		// Go back to start
		_inst_intStep := 0;
END_CASE

M_Enable := _bResult;
intEnableStep := _inst_intStep;
END_METHOD

(* This method should explicitly check the enable status of the device.
	Once the enable status is known, this method should return TRUE.
	If this method fails, P_bEnabled should be set to FALSE since the device
	is not absolutely known to still be enabled. *)
METHOD M_GetEnableStatus : BOOL
VAR_OUTPUT
	(* This should return TRUE if the device is explicitly known to be
		enabled, or FALSE otherwise. *)
	bEnabled	: BOOL;
END_VAR
VAR CONSTANT
	_strCOMMAND_NAME : T_MaxString	:= 'GetEnableStatus'; // Name of the API method
	_timeCOMMAND_TIMEOUT : TIME		:= T#5S; // Max time to receive API response
	_strSTART_MSG : T_MaxString		:= 'Getting enable status'; // Prints when method starts
	_strEND_MSG : T_MaxString		:= 'Received enable status'; // Prints when method finishes
	_udintERROR_ID : UDINT			:= E_ApiDeviceError.FailedToGetEnableStatus; // Error ID to set if command fails
	_strERROR_MSG : T_MaxString		:= 'Failed to get enable status!'; // Error message to set if command fails
END_VAR
VAR_INST
	_inst_arrParams: T_ApiParameterList; // Parameters array
	_inst_arrOutputs: T_ApiParameterList; // Outputs array
	_inst_strRet: T_ApiParamValue; // Return string from the router
	_inst_intStep: INT; // Current method step
	_inst_fbParams: FB_ApiParamBuilder; // Parameter builder FB
END_VAR
VAR
	_bComplete: BOOL; // True if the routing finishes
	_intRet: INT; // Return string converted to an integer
	_bResult : BOOL; // Output of the method
	_pArgs: PVOID; // Arguments pointer
END_VAR
_bResult := FALSE;

// Recover from premature stop
bGetEnableStatusBusy := TRUE;
_inst_intStep := intGetEnableStatusStep;

// Steps
CASE _inst_intStep OF
	0: // Wait for no error and router not busy
		IF NOT THIS^.P_bError AND NOT bRouterBusy THEN
			bRouterBusy := TRUE;
			_inst_intStep := _inst_intStep + 10;
		END_IF
		
	10: // Initialize parameters
		THIS^.M_LogMessage(_strSTART_MSG);
		_inst_fbParams.M_ClearParameters();
		_pArgs := _inst_fbParams.M_AddEmptyStruct('args');
		_inst_fbParams.M_OutputToParameterList(_inst_arrParams);
		_inst_intStep := _inst_intStep + 10;
		
	20: // Route the command
		_bComplete := M_RouterHelper(
			_in_strMethodName := _strCOMMAND_NAME, 
			_in_timeTimeout := _timeCOMMAND_TIMEOUT,
			_inout_arrParams := _inst_arrParams,
			_inout_arrOutputs := _inst_arrOutputs,
			_out_strReturnValue=>_inst_strRet);
		
		// If route completed, move to next step
		IF _bComplete THEN
			_inst_intStep := _inst_intStep + 10;
			bRouterBusy := FALSE;
		ELSIF THIS^.P_bError THEN
			_inst_intStep := 0;
			bRouterBusy := FALSE;
		END_IF
		
	30: // Parse results
		_intRet := STRING_TO_INT(_inst_strRet);
		IF _intRet > 0 THEN
			_bResult := TRUE;
			THIS^.M_LogMessage(_strEND_MSG);
			_inst_fbParams.M_LoadFromParameterList(_inst_arrOutputs);
			THIS^.bEnabled := _inst_fbParams.M_ParseBool(
				_inst_fbParams.M_GetParameter('enabled'));
			bEnabled := THIS^.bEnabled;
			
		// Set error if command failed
		ELSE
			THIS^.M_SetError(_udintERROR_ID, _strERROR_MSG);
		END_IF
		
		// Go back to start
		_inst_intStep := 0;
END_CASE

M_GetEnableStatus := _bResult;
intGetEnableStatusStep := _inst_intStep;
END_METHOD

(* This property should be TRUE while any method in this interface is actively
	executing, or FALSE otherwise. *)
PROPERTY P_bEnableBusy : BOOL
GET
P_bEnableBusy := bRouterBusy;
END_GET
END_PROPERTY

(* This should be set to TRUE if M_Enable is successful or M_GetEnableStatus
	determines the device to be enabled, and set to FALSE if M_Disable is
	called at all, M_GetEnableStatus fails, or M_GetEnableStatus determines
	the device to be not enabled. *)
PROPERTY P_bEnabled : BOOL
GET
P_bEnabled := bEnabled;
END_GET
END_PROPERTY

(* This method should explicitly check the power status of the device.
	Once the power status is known, this method should return TRUE.
	If this method fails, P_bPoweredOn should be set to FALSE since the device
	is not absolutely known to still be powered on. *)
METHOD M_GetPowerStatus : BOOL
VAR_OUTPUT
	(* This should return TRUE if the device is explicitly known to be
		powered on, or FALSE otherwise. *)
	bPoweredOn	: BOOL;
END_VAR
VAR CONSTANT
	_strCOMMAND_NAME : T_MaxString	:= 'GetPowerStatus'; // Name of the API method
	_timeCOMMAND_TIMEOUT : TIME		:= T#5S; // Max time to receive API response
	_strSTART_MSG : T_MaxString		:= 'Getting power status'; // Prints when method starts
	_strEND_MSG : T_MaxString		:= 'Received power status'; // Prints when method finishes
	_udintERROR_ID : UDINT			:= E_ApiDeviceError.FailedToGetPowerStatus; // Error ID to set if command fails
	_strERROR_MSG : T_MaxString		:= 'Failed to get power status!'; // Error message to set if command fails
END_VAR
VAR_INST
	_inst_arrParams: T_ApiParameterList; // Parameters array
	_inst_arrOutputs: T_ApiParameterList; // Outputs array
	_inst_strRet: T_ApiParamValue; // Return string from the router
	_inst_intStep: INT; // Current method step
	_inst_fbParams: FB_ApiParamBuilder; // Parameter builder FB
END_VAR
VAR
	_bComplete: BOOL; // True if the routing finishes
	_intRet: INT; // Return string converted to an integer
	_bResult : BOOL; // Output of the method
	_pArgs: PVOID; // Arguments pointer
END_VAR
_bResult := FALSE;

// Recover from premature stop
bGetPowerStatusBusy := TRUE;
_inst_intStep := intGetPowerStatusStep;

// Steps
CASE _inst_intStep OF
	0: // Wait for no error and router not busy
		IF NOT THIS^.P_bError AND NOT bRouterBusy THEN
			bRouterBusy := TRUE;
			_inst_intStep := _inst_intStep + 10;
		END_IF
		
	10: // Initialize parameters
		THIS^.M_LogMessage(_strSTART_MSG);
		_inst_fbParams.M_ClearParameters();
		_pArgs := _inst_fbParams.M_AddEmptyStruct('args');
		_inst_fbParams.M_OutputToParameterList(_inst_arrParams);
		_inst_intStep := _inst_intStep + 10;
		
	20: // Route the command
		_bComplete := M_RouterHelper(
			_in_strMethodName := _strCOMMAND_NAME, 
			_in_timeTimeout := _timeCOMMAND_TIMEOUT,
			_inout_arrParams := _inst_arrParams,
			_inout_arrOutputs := _inst_arrOutputs,
			_out_strReturnValue=>_inst_strRet);
		
		// If route completed, move to next step
		IF _bComplete THEN
			_inst_intStep := _inst_intStep + 10;
			bRouterBusy := FALSE;
		ELSIF THIS^.P_bError THEN
			_inst_intStep := 0;
			bRouterBusy := FALSE;
		END_IF
		
	30: // Parse results
		_intRet := STRING_TO_INT(_inst_strRet);
		IF _intRet > 0 THEN
			_bResult := TRUE;
			THIS^.M_LogMessage(_strEND_MSG);
			_inst_fbParams.M_LoadFromParameterList(_inst_arrOutputs);
			THIS^.bPoweredOn := _inst_fbParams.M_ParseBool(
				_inst_fbParams.M_GetParameter('poweredOn'));
			bPoweredOn := THIS^.bPoweredOn;
			
		// Set error if command failed
		ELSE
			THIS^.M_SetError(_udintERROR_ID, _strERROR_MSG);
		END_IF
		
		// Go back to start
		_inst_intStep := 0;
END_CASE

M_GetPowerStatus := _bResult;
intGetPowerStatusStep := _inst_intStep;
END_METHOD

(* This method should de-energize the device and then return TRUE once
	successful. P_bPoweredOn should be set to FALSE immediately when this is
	called unless the device is explicitly known to still be powered on. *)
METHOD M_PowerOff : BOOL
VAR CONSTANT
	_strCOMMAND_NAME : T_MaxString	:= 'PowerOff'; // Name of the API method
	_timeCOMMAND_TIMEOUT : TIME		:= T#30S; // Max time to receive API response
	_strSTART_MSG : T_MaxString		:= 'Powering off'; // Prints when method starts
	_strEND_MSG : T_MaxString		:= 'Powered off'; // Prints when method finishes
	_udintERROR_ID : UDINT			:= E_ApiDeviceError.FailedToPowerOff; // Error ID to set if command fails
	_strERROR_MSG : T_MaxString		:= 'Failed to power off!'; // Error message to set if command fails
END_VAR
VAR_INST
	_inst_arrParams: T_ApiParameterList; // Parameters array
	_inst_arrOutputs: T_ApiParameterList; // Outputs array
	_inst_strRet: T_ApiParamValue; // Return string from the router
	_inst_intStep: INT; // Current method step
	_inst_fbParams: FB_ApiParamBuilder; // Parameter builder FB
END_VAR
VAR
	_bComplete: BOOL; // True if the routing finishes
	_intRet: INT; // Return string converted to an integer
	_bResult : BOOL; // Output of the method
	_pArgs: PVOID; // Arguments pointer
END_VAR
_bResult := FALSE;

// Recover from premature stop
bPowerOffBusy := TRUE;
_inst_intStep := intPowerOffStep;

// Steps
CASE _inst_intStep OF
	0: // Wait for no error and router not busy
		IF NOT THIS^.P_bError AND NOT bRouterBusy THEN
			bRouterBusy := TRUE;
			_inst_intStep := _inst_intStep + 10;
		END_IF
		
	10: // Initialize parameters
		THIS^.M_LogMessage(_strSTART_MSG);
		_inst_fbParams.M_ClearParameters();
		_pArgs := _inst_fbParams.M_AddEmptyStruct('args');
		_inst_fbParams.M_OutputToParameterList(_inst_arrParams);
		_inst_intStep := _inst_intStep + 10;
		
	20: // Route the command
		_bComplete := M_RouterHelper(
			_in_strMethodName := _strCOMMAND_NAME, 
			_in_timeTimeout := _timeCOMMAND_TIMEOUT,
			_inout_arrParams := _inst_arrParams,
			_inout_arrOutputs := _inst_arrOutputs,
			_out_strReturnValue=>_inst_strRet);
		
		// If route completed, move to next step
		IF _bComplete THEN
			_inst_intStep := _inst_intStep + 10;
			bRouterBusy := FALSE;
		ELSIF THIS^.P_bError THEN
			_inst_intStep := 0;
			bRouterBusy := FALSE;
		END_IF
		
	30: // Parse results
		_intRet := STRING_TO_INT(_inst_strRet);
		IF _intRet > 0 THEN
			_bResult := TRUE;
			THIS^.M_LogMessage(_strEND_MSG);
			_inst_fbParams.M_LoadFromParameterList(_inst_arrOutputs);
			bPoweredOn := FALSE;
			
		// Set error if command failed
		ELSE
			THIS^.M_SetError(_udintERROR_ID, _strERROR_MSG);
		END_IF
		
		// Go back to start
		_inst_intStep := 0;
END_CASE

M_PowerOff := _bResult;
intPowerOffStep := _inst_intStep;
END_METHOD

(* This method should energize the device and then return TRUE and set
	P_bPoweredOn to TRUE once successful. *)
METHOD M_PowerOn : BOOL
VAR CONSTANT
	_strCOMMAND_NAME : T_MaxString	:= 'PowerOn'; // Name of the API method
	_timeCOMMAND_TIMEOUT : TIME		:= T#30S; // Max time to receive API response
	_strSTART_MSG : T_MaxString		:= 'Powering on'; // Prints when method starts
	_strEND_MSG : T_MaxString		:= 'Powered on'; // Prints when method finishes
	_udintERROR_ID : UDINT			:= E_ApiDeviceError.FailedToPowerOn; // Error ID to set if command fails
	_strERROR_MSG : T_MaxString		:= 'Failed to power on!'; // Error message to set if command fails
END_VAR
VAR_INST
	_inst_arrParams: T_ApiParameterList; // Parameters array
	_inst_arrOutputs: T_ApiParameterList; // Outputs array
	_inst_strRet: T_ApiParamValue; // Return string from the router
	_inst_intStep: INT; // Current method step
	_inst_fbParams: FB_ApiParamBuilder; // Parameter builder FB
END_VAR
VAR
	_bComplete: BOOL; // True if the routing finishes
	_intRet: INT; // Return string converted to an integer
	_bResult : BOOL; // Output of the method
	_pArgs: PVOID; // Arguments pointer
END_VAR
_bResult := FALSE;

// Recover from premature stop
bPowerOnBusy := TRUE;
_inst_intStep := intPowerOnStep;

// Steps
CASE _inst_intStep OF
	0: // Wait for no error and router not busy
		IF NOT THIS^.P_bError AND NOT bRouterBusy THEN
			bRouterBusy := TRUE;
			_inst_intStep := _inst_intStep + 10;
		END_IF
		
	10: // Initialize parameters
		THIS^.M_LogMessage(_strSTART_MSG);
		_inst_fbParams.M_ClearParameters();
		_pArgs := _inst_fbParams.M_AddEmptyStruct('args');
		_inst_fbParams.M_AddStructMember(_pArgs, 'scannerName', in_strScannerName);
		_inst_fbParams.M_OutputToParameterList(_inst_arrParams);
		_inst_intStep := _inst_intStep + 10;
		
	20: // Route the command
		_bComplete := M_RouterHelper(
			_in_strMethodName := _strCOMMAND_NAME, 
			_in_timeTimeout := _timeCOMMAND_TIMEOUT,
			_inout_arrParams := _inst_arrParams,
			_inout_arrOutputs := _inst_arrOutputs,
			_out_strReturnValue=>_inst_strRet);
		
		// If route completed, move to next step
		IF _bComplete THEN
			_inst_intStep := _inst_intStep + 10;
			bRouterBusy := FALSE;
		ELSIF THIS^.P_bError THEN
			_inst_intStep := 0;
			bRouterBusy := FALSE;
		END_IF
		
	30: // Parse results
		_intRet := STRING_TO_INT(_inst_strRet);
		IF _intRet > 0 THEN
			_bResult := TRUE;
			THIS^.M_LogMessage(_strEND_MSG);
			_inst_fbParams.M_LoadFromParameterList(_inst_arrOutputs);
			bPoweredOn := TRUE;
			
		// Set error if command failed
		ELSE
			THIS^.M_SetError(_udintERROR_ID, _strERROR_MSG);
		END_IF
		
		// Go back to start
		_inst_intStep := 0;
END_CASE

M_PowerOn := _bResult;
intPowerOnStep := _inst_intStep;
END_METHOD

(* This property should be TRUE while any method in this interface is actively
	executing, or FALSE otherwise. *)
PROPERTY P_bPowerBusy : BOOL
GET
P_bPowerBusy := bRouterBusy;
END_GET
END_PROPERTY

(* This should be set to TRUE if M_PowerOn is successful or if M_GetPowerStatus
	determines that the device is powered on. Otherwise, this should be FALSE. *)
PROPERTY P_bPoweredOn : BOOL
GET
P_bPoweredOn := bPoweredOn;
END_GET
END_PROPERTY

(* This method should explicitly get the current program loaded on the device.
	If the current program is successfully gotten, this method should return
	TRUE and set P_strCurrentProgram and strCurrentProgram to the gotten
	program name. If this method fails, both should be set to empty strings. *)
METHOD M_GetCurrentProgram : BOOL
VAR_OUTPUT
	(* This should be set to the name of the currently loaded program if
		the method was successful, or a blank string otherwise. *)
	strCurrentProgram	: Sensata_Common.T_MaxString;
END_VAR
VAR CONSTANT
	_strCOMMAND_NAME : T_MaxString	:= 'GetCurrentProgram'; // Name of the API method
	_timeCOMMAND_TIMEOUT : TIME		:= T#10S; // Max time to receive API response
	_strSTART_MSG : T_MaxString		:= 'Getting current program'; // Prints when method starts
	_strEND_MSG : T_MaxString		:= 'Received current program'; // Prints when method finishes
	_udintERROR_ID : UDINT			:= E_ApiDeviceError.FailedToGetCurrentProgram; // Error ID to set if command fails
	_strERROR_MSG : T_MaxString		:= 'Failed to get current program!'; // Error message to set if command fails
END_VAR
VAR_INST
	_inst_arrParams: T_ApiParameterList; // Parameters array
	_inst_arrOutputs: T_ApiParameterList; // Outputs array
	_inst_strRet: T_ApiParamValue; // Return string from the router
	_inst_intStep: INT; // Current method step
	_inst_fbParams: FB_ApiParamBuilder; // Parameter builder FB
END_VAR
VAR
	_bComplete: BOOL; // True if the routing finishes
	_intRet: INT; // Return string converted to an integer
	_bResult : BOOL; // Output of the method
	_pArgs: PVOID; // Arguments pointer
END_VAR
_bResult := FALSE;

// Recover from premature stop
bGetCurrentProgramBusy := TRUE;
_inst_intStep := intGetCurrentProgramStep;

// Steps
CASE _inst_intStep OF
	0: // Wait for no error and router not busy
		IF NOT THIS^.P_bError AND NOT bRouterBusy THEN
			bRouterBusy := TRUE;
			_inst_intStep := _inst_intStep + 10;
		END_IF
		
	10: // Initialize parameters
		THIS^.M_LogMessage(_strSTART_MSG);
		_inst_fbParams.M_ClearParameters();
		_pArgs := _inst_fbParams.M_AddEmptyStruct('args');
		_inst_fbParams.M_OutputToParameterList(_inst_arrParams);
		_inst_intStep := _inst_intStep + 10;
		
	20: // Route the command
		_bComplete := M_RouterHelper(
			_in_strMethodName := _strCOMMAND_NAME, 
			_in_timeTimeout := _timeCOMMAND_TIMEOUT,
			_inout_arrParams := _inst_arrParams,
			_inout_arrOutputs := _inst_arrOutputs,
			_out_strReturnValue=>_inst_strRet);
		
		// If route completed, move to next step
		IF _bComplete THEN
			_inst_intStep := _inst_intStep + 10;
			bRouterBusy := FALSE;
		ELSIF THIS^.P_bError THEN
			_inst_intStep := 0;
			bRouterBusy := FALSE;
		END_IF
		
	30: // Parse results
		_intRet := STRING_TO_INT(_inst_strRet);
		IF _intRet > 0 THEN
			_bResult := TRUE;
			THIS^.M_LogMessage(_strEND_MSG);
			_inst_fbParams.M_LoadFromParameterList(_inst_arrOutputs);
			THIS^.strLoadedProgram := _inst_fbParams.M_ParseString(
				_inst_fbParams.M_GetParameter('programName'));
			strCurrentProgram := THIS^.strLoadedProgram;
			
		// Set error if command failed
		ELSE
			THIS^.M_SetError(_udintERROR_ID, _strERROR_MSG);
		END_IF
		
		// Go back to start
		_inst_intStep := 0;
END_CASE

M_GetCurrentProgram := _bResult;
intGetCurrentProgramStep := _inst_intStep;
END_METHOD

(* This method should explicitly check the program state of the device.
	Once the program state is known, this method should return TRUE and set
	P_enumProgramState and enumProgramState to the relevant E_ProgramState
	value, else it should set both to E_ProgramState.Unknown. *)
METHOD M_GetProgramState : BOOL
VAR_OUTPUT
	(* If the program state is successfully gotten, this should be set to
		the relevant E_ProgramState value. If this method fails, this should
		be set to E_ProgramState.Unknown. *)
	enumProgramState	: Sensata_Common.E_ProgramState;
END_VAR
VAR CONSTANT
	_strCOMMAND_NAME : T_MaxString	:= 'GetControlState'; // Name of the API method
	_timeCOMMAND_TIMEOUT : TIME		:= T#10S; // Max time to receive API response
	_strSTART_MSG : T_MaxString		:= 'Getting program state'; // Prints when method starts
	_strEND_MSG : T_MaxString		:= 'Received program state'; // Prints when method finishes
	_udintERROR_ID : UDINT			:= E_ApiDeviceError.FailedToGetProgramState; // Error ID to set if command fails
	_strERROR_MSG : T_MaxString		:= 'Failed to get program state!'; // Error message to set if command fails
END_VAR
VAR_INST
	_inst_arrParams: T_ApiParameterList; // Parameters array
	_inst_arrOutputs: T_ApiParameterList; // Outputs array
	_inst_strRet: T_ApiParamValue; // Return string from the router
	_inst_intStep: INT; // Current method step
	_inst_fbParams: FB_ApiParamBuilder; // Parameter builder FB
END_VAR
VAR
	_bComplete: BOOL; // True if the routing finishes
	_intRet: INT; // Return string converted to an integer
	_bResult : BOOL; // Output of the method
	_pArgs: PVOID; // Arguments pointer
	dintControlState: DINT; // Current program state
END_VAR
_bResult := FALSE;

// Recover from premature stop
bGetProgramStateBusy := TRUE;
_inst_intStep := intGetProgramStateStep;

// Steps
CASE _inst_intStep OF
	0: // Wait for no error and router not busy
		IF NOT THIS^.P_bError AND NOT bRouterBusy THEN
			bRouterBusy := TRUE;
			_inst_intStep := _inst_intStep + 10;
		END_IF
		
	10: // Initialize parameters
		THIS^.M_LogMessage(_strSTART_MSG);
		_inst_fbParams.M_ClearParameters();
		_pArgs := _inst_fbParams.M_AddEmptyStruct('args');
		_inst_fbParams.M_OutputToParameterList(_inst_arrParams);
		_inst_intStep := _inst_intStep + 10;
		
	20: // Route the command
		_bComplete := M_RouterHelper(
			_in_strMethodName := _strCOMMAND_NAME, 
			_in_timeTimeout := _timeCOMMAND_TIMEOUT,
			_inout_arrParams := _inst_arrParams,
			_inout_arrOutputs := _inst_arrOutputs,
			_out_strReturnValue=>_inst_strRet);
		
		// If route completed, move to next step
		IF _bComplete THEN
			_inst_intStep := _inst_intStep + 10;
			bRouterBusy := FALSE;
		ELSIF THIS^.P_bError THEN
			_inst_intStep := 0;
			bRouterBusy := FALSE;
		END_IF
		
	30: // Parse results
		_intRet := STRING_TO_INT(_inst_strRet);
		IF _intRet > 0 THEN
			_bResult := TRUE;
			THIS^.M_LogMessage(_strEND_MSG);
			_inst_fbParams.M_LoadFromParameterList(_inst_arrOutputs);
			dintControlState := _inst_fbParams.M_ParseInt(_inst_fbParams.M_GetParameter('state'));
			CASE dintControlState OF
				0: enumProgramState := E_ProgramState.Unknown;
				1: enumProgramState := E_ProgramState.Stopped;
				2: enumProgramState := E_ProgramState.Running;
				3: enumProgramState := E_ProgramState.Paused;
			ELSE
				enumProgramState := E_ProgramState.Unknown;
			END_CASE
			THIS^.enumProgramState := enumProgramState;
			
		// Set error if command failed
		ELSE
			THIS^.M_SetError(_udintERROR_ID, _strERROR_MSG);
		END_IF
		
		// Go back to start
		_inst_intStep := 0;
END_CASE

M_GetProgramState := _bResult;
intGetProgramStateStep := _inst_intStep;
END_METHOD

(* This method should load a new program onto the device, and then return TRUE
	once program loading is completed. Once this method begins the program loading
	process, P_strCurrentProgram should be cleared unless it is still explicitly
	known to be loaded. *)
METHOD M_LoadProgram : BOOL
VAR_INPUT
END_VAR
VAR CONSTANT
	_strCOMMAND_NAME : T_MaxString	:= 'LoadProgram'; // Name of the API method
	_timeCOMMAND_TIMEOUT : TIME		:= T#30S; // Max time to receive API response
	_strSTART_MSG : T_MaxString		:= 'Loading program'; // Prints when method starts
	_strEND_MSG : T_MaxString		:= 'Loaded program'; // Prints when method finishes
	_udintERROR_ID : UDINT			:= E_ApiDeviceError.FailedToLoadProgram; // Error ID to set if command fails
	_strERROR_MSG : T_MaxString		:= 'Failed to load program!'; // Error message to set if command fails
END_VAR
VAR_INST
	_inst_arrParams: T_ApiParameterList; // Parameters array
	_inst_arrOutputs: T_ApiParameterList; // Outputs array
	_inst_strRet: T_ApiParamValue; // Return string from the router
	_inst_intStep: INT; // Current method step
	_inst_fbParams: FB_ApiParamBuilder; // Parameter builder FB
END_VAR
VAR
	_bComplete: BOOL; // True if the routing finishes
	_intRet: INT; // Return string converted to an integer
	_bResult : BOOL; // Output of the method
	_pArgs: PVOID; // Arguments pointer
END_VAR
_bResult := FALSE;

// Recover from premature stop
bLoadProgramBusy := TRUE;
_inst_intStep := intLoadProgramStep;

// Steps
CASE _inst_intStep OF
	0: // Wait for no error and router not busy
		IF NOT THIS^.P_bError AND NOT bRouterBusy THEN
			bRouterBusy := TRUE;
			_inst_intStep := _inst_intStep + 10;
		END_IF
		
	10: // Initialize parameters
		THIS^.M_LogMessage(_strSTART_MSG);
		_inst_fbParams.M_ClearParameters();
		_pArgs := _inst_fbParams.M_AddEmptyStruct('args');
		_inst_fbParams.M_AddStructMember(_pArgs, 'filename', in_strProgramName);
		_inst_fbParams.M_OutputToParameterList(_inst_arrParams);
		_inst_intStep := _inst_intStep + 10;
		
	20: // Route the command
		_bComplete := M_RouterHelper(
			_in_strMethodName := _strCOMMAND_NAME, 
			_in_timeTimeout := _timeCOMMAND_TIMEOUT,
			_inout_arrParams := _inst_arrParams,
			_inout_arrOutputs := _inst_arrOutputs,
			_out_strReturnValue=>_inst_strRet);
		
		// If route completed, move to next step
		IF _bComplete THEN
			_inst_intStep := _inst_intStep + 10;
			bRouterBusy := FALSE;
		ELSIF THIS^.P_bError THEN
			_inst_intStep := 0;
			bRouterBusy := FALSE;
		END_IF
		
	30: // Parse results
		_intRet := STRING_TO_INT(_inst_strRet);
		IF _intRet > 0 THEN
			_bResult := TRUE;
			THIS^.M_LogMessage(_strEND_MSG);
			_inst_fbParams.M_LoadFromParameterList(_inst_arrOutputs);
			strLoadedProgram := '';
			
		// Set error if command failed
		ELSE
			THIS^.M_SetError(_udintERROR_ID, _strERROR_MSG);
		END_IF
		
		// Go back to start
		_inst_intStep := 0;
END_CASE

M_LoadProgram := _bResult;
intLoadProgramStep := _inst_intStep;
END_METHOD

(* This program should move to the program state from whatever state it was in
	to the Paused state, and then return TRUE once successful. If the program
	state is Stopped, this method should return TRUE but keep the current state
	as Stopped, since Paused at the beginning at the program is equivalent to
	being Stopped. *)
METHOD M_PauseProgram : BOOL
VAR CONSTANT
	_strCOMMAND_NAME : T_MaxString	:= 'PauseProgram'; // Name of the API method
	_timeCOMMAND_TIMEOUT : TIME		:= T#30S; // Max time to receive API response
	_strSTART_MSG : T_MaxString		:= 'Pausing program'; // Prints when method starts
	_strEND_MSG : T_MaxString		:= 'Paused program'; // Prints when method finishes
	_udintERROR_ID : UDINT			:= E_ApiDeviceError.FailedToPauseProgram; // Error ID to set if command fails
	_strERROR_MSG : T_MaxString		:= 'Failed to pause program!'; // Error message to set if command fails
END_VAR
VAR_INST
	_inst_arrParams: T_ApiParameterList; // Parameters array
	_inst_arrOutputs: T_ApiParameterList; // Outputs array
	_inst_strRet: T_ApiParamValue; // Return string from the router
	_inst_intStep: INT; // Current method step
	_inst_fbParams: FB_ApiParamBuilder; // Parameter builder FB
END_VAR
VAR
	_bComplete: BOOL; // True if the routing finishes
	_intRet: INT; // Return string converted to an integer
	_bResult : BOOL; // Output of the method
	_pArgs: PVOID; // Arguments pointer
END_VAR
_bResult := FALSE;

// Recover from premature stop
bPauseProgramBusy := TRUE;
_inst_intStep := intPauseProgramStep;

// Steps
CASE _inst_intStep OF
	0: // Wait for no error and router not busy
		IF NOT THIS^.P_bError AND NOT bRouterBusy THEN
			bRouterBusy := TRUE;
			_inst_intStep := _inst_intStep + 10;
		END_IF
		
	10: // Initialize parameters
		THIS^.M_LogMessage(_strSTART_MSG);
		_inst_fbParams.M_ClearParameters();
		_pArgs := _inst_fbParams.M_AddEmptyStruct('args');
		_inst_fbParams.M_OutputToParameterList(_inst_arrParams);
		_inst_intStep := _inst_intStep + 10;
		
	20: // Route the command
		_bComplete := M_RouterHelper(
			_in_strMethodName := _strCOMMAND_NAME, 
			_in_timeTimeout := _timeCOMMAND_TIMEOUT,
			_inout_arrParams := _inst_arrParams,
			_inout_arrOutputs := _inst_arrOutputs,
			_out_strReturnValue=>_inst_strRet);
		
		// If route completed, move to next step
		IF _bComplete THEN
			_inst_intStep := _inst_intStep + 10;
			bRouterBusy := FALSE;
		ELSIF THIS^.P_bError THEN
			_inst_intStep := 0;
			bRouterBusy := FALSE;
		END_IF
		
	30: // Parse results
		_intRet := STRING_TO_INT(_inst_strRet);
		IF _intRet > 0 THEN
			_bResult := TRUE;
			THIS^.M_LogMessage(_strEND_MSG);
			_inst_fbParams.M_LoadFromParameterList(_inst_arrOutputs);
			enumProgramState := E_ProgramState.Paused;
			
		// Set error if command failed
		ELSE
			THIS^.M_SetError(_udintERROR_ID, _strERROR_MSG);
		END_IF
		
		// Go back to start
		_inst_intStep := 0;
END_CASE

M_PauseProgram := _bResult;
intPauseProgramStep := _inst_intStep;
END_METHOD

(* This should move the program state from whatever state it is in to the
	Running state, and then return TRUE once successful. Starting from the
	Paused state should always continue execution from whatever point the
	program was at when the program was initially paused. *)
METHOD M_StartProgram : BOOL
VAR CONSTANT
	_strCOMMAND_NAME : T_MaxString	:= 'StartProgram'; // Name of the API method
	_timeCOMMAND_TIMEOUT : TIME		:= T#30S; // Max time to receive API response
	_strSTART_MSG : T_MaxString		:= 'Starting program'; // Prints when method starts
	_strEND_MSG : T_MaxString		:= 'Started program'; // Prints when method finishes
	_udintERROR_ID : UDINT			:= E_ApiDeviceError.FailedToStartProgram; // Error ID to set if command fails
	_strERROR_MSG : T_MaxString		:= 'Failed to start program!'; // Error message to set if command fails
END_VAR
VAR_INST
	_inst_arrParams: T_ApiParameterList; // Parameters array
	_inst_arrOutputs: T_ApiParameterList; // Outputs array
	_inst_strRet: T_ApiParamValue; // Return string from the router
	_inst_intStep: INT; // Current method step
	_inst_fbParams: FB_ApiParamBuilder; // Parameter builder FB
END_VAR
VAR
	_bComplete: BOOL; // True if the routing finishes
	_intRet: INT; // Return string converted to an integer
	_bResult : BOOL; // Output of the method
	_pArgs: PVOID; // Arguments pointer
END_VAR
_bResult := FALSE;

// Recover from premature stop
bStartProgramBusy := TRUE;
_inst_intStep := intStartProgramStep;

// Steps
CASE _inst_intStep OF
	0: // Wait for no error and router not busy
		IF NOT THIS^.P_bError AND NOT bRouterBusy THEN
			bRouterBusy := TRUE;
			_inst_intStep := _inst_intStep + 10;
		END_IF
		
	10: // Initialize parameters
		THIS^.M_LogMessage(_strSTART_MSG);
		_inst_fbParams.M_ClearParameters();
		_pArgs := _inst_fbParams.M_AddEmptyStruct('args');
		_inst_fbParams.M_OutputToParameterList(_inst_arrParams);
		_inst_intStep := _inst_intStep + 10;
		
	20: // Route the command
		_bComplete := M_RouterHelper(
			_in_strMethodName := _strCOMMAND_NAME, 
			_in_timeTimeout := _timeCOMMAND_TIMEOUT,
			_inout_arrParams := _inst_arrParams,
			_inout_arrOutputs := _inst_arrOutputs,
			_out_strReturnValue=>_inst_strRet);
		
		// If route completed, move to next step
		IF _bComplete THEN
			_inst_intStep := _inst_intStep + 10;
			bRouterBusy := FALSE;
		ELSIF THIS^.P_bError THEN
			_inst_intStep := 0;
			bRouterBusy := FALSE;
		END_IF
		
	30: // Parse results
		_intRet := STRING_TO_INT(_inst_strRet);
		IF _intRet > 0 THEN
			_bResult := TRUE;
			THIS^.M_LogMessage(_strEND_MSG);
			_inst_fbParams.M_LoadFromParameterList(_inst_arrOutputs);
			enumProgramState := E_ProgramState.Running;
			
		// Set error if command failed
		ELSE
			THIS^.M_SetError(_udintERROR_ID, _strERROR_MSG);
		END_IF
		
		// Go back to start
		_inst_intStep := 0;
END_CASE

M_StartProgram := _bResult;
intStartProgramStep := _inst_intStep;
END_METHOD

(* This should change the program state from whatever state it was in to the
	Stopped state and then return TRUE. Moving to the Stopped state should
	always reset the program execution back to the beginning. *)
METHOD M_StopProgram : BOOL
VAR CONSTANT
	_strCOMMAND_NAME : T_MaxString	:= 'StopProgram'; // Name of the API method
	_timeCOMMAND_TIMEOUT : TIME		:= T#30S; // Max time to receive API response
	_strSTART_MSG : T_MaxString		:= 'Stopping'; // Prints when method starts
	_strEND_MSG : T_MaxString		:= 'Stopped'; // Prints when method finishes
	_udintERROR_ID : UDINT			:= E_ApiDeviceError.FailedToStopProgram; // Error ID to set if command fails
	_strERROR_MSG : T_MaxString		:= 'Failed to stop program!'; // Error message to set if command fails
END_VAR
VAR_INST
	_inst_arrParams: T_ApiParameterList; // Parameters array
	_inst_arrOutputs: T_ApiParameterList; // Outputs array
	_inst_strRet: T_ApiParamValue; // Return string from the router
	_inst_intStep: INT; // Current method step
	_inst_fbParams: FB_ApiParamBuilder; // Parameter builder FB
END_VAR
VAR
	_bComplete: BOOL; // True if the routing finishes
	_intRet: INT; // Return string converted to an integer
	_bResult : BOOL; // Output of the method
	_pArgs: PVOID; // Arguments pointer
END_VAR
_bResult := FALSE;

// Recover from premature stop
bStopProgramBusy := TRUE;
_inst_intStep := intStopProgramStep;

// Steps
CASE _inst_intStep OF
	0: // Wait for no error and router not busy
		IF NOT THIS^.P_bError AND NOT bRouterBusy THEN
			bRouterBusy := TRUE;
			_inst_intStep := _inst_intStep + 10;
		END_IF
		
	10: // Initialize parameters
		THIS^.M_LogMessage(_strSTART_MSG);
		_inst_fbParams.M_ClearParameters();
		_pArgs := _inst_fbParams.M_AddEmptyStruct('args');
		_inst_fbParams.M_OutputToParameterList(_inst_arrParams);
		_inst_intStep := _inst_intStep + 10;
		
	20: // Route the command
		_bComplete := M_RouterHelper(
			_in_strMethodName := _strCOMMAND_NAME, 
			_in_timeTimeout := _timeCOMMAND_TIMEOUT,
			_inout_arrParams := _inst_arrParams,
			_inout_arrOutputs := _inst_arrOutputs,
			_out_strReturnValue=>_inst_strRet);
		
		// If route completed, move to next step
		IF _bComplete THEN
			_inst_intStep := _inst_intStep + 10;
			bRouterBusy := FALSE;
		ELSIF THIS^.P_bError THEN
			_inst_intStep := 0;
			bRouterBusy := FALSE;
		END_IF
		
	30: // Parse results
		_intRet := STRING_TO_INT(_inst_strRet);
		IF _intRet > 0 THEN
			_bResult := TRUE;
			THIS^.M_LogMessage(_strEND_MSG);
			_inst_fbParams.M_LoadFromParameterList(_inst_arrOutputs);
			enumProgramState := E_ProgramState.Stopped;
			
		// Set error if command failed
		ELSE
			THIS^.M_SetError(_udintERROR_ID, _strERROR_MSG);
		END_IF
		
		// Go back to start
		_inst_intStep := 0;
END_CASE

M_StopProgram := _bResult;
intStopProgramStep := _inst_intStep;
END_METHOD

(* This property should be TRUE while any method in this interface is actively
	executing, or FALSE otherwise. *)
PROPERTY P_bProgramControlBusy : BOOL
GET
P_bProgramControlBusy := bRouterBusy;
END_GET
END_PROPERTY

(* The current E_ProgramState value of the device. This should be reset to
	E_ProgramState.Unknown if any methods in this interface interact with the
	device but fail. *)
PROPERTY P_enumProgramState : Sensata_Common.E_ProgramState
GET
P_enumProgramState := enumProgramState;
END_GET
END_PROPERTY

(* The value of the currently loaded program. This should only be set by
	M_LoadProgram or M_GetCurrentProgram, and set to a blank string if either
	fail. *)
PROPERTY P_strCurrentProgram : Sensata_Common.T_MaxString
GET
P_strCurrentProgram := strLoadedProgram;
END_GET
END_PROPERTY

(* This method should establish any external connections required to use the
	functions of the device, and return TRUE and set P_bConnected to TRUE once
	connected. *)
METHOD M_Reset : BOOL
VAR CONSTANT
	_strCOMMAND_NAME : T_MaxString	:= 'Reset'; // Name of the API method
	_timeCOMMAND_TIMEOUT : TIME		:= T#30S; // Max time to receive API response
	_strSTART_MSG : T_MaxString		:= 'Resetting'; // Prints when method starts
	_strEND_MSG : T_MaxString		:= 'Reset'; // Prints when method finishes
	_udintERROR_ID : UDINT			:= E_ApiDeviceError.FailedToReset; // Error ID to set if command fails
	_strERROR_MSG : T_MaxString		:= 'Failed to reset!'; // Error message to set if command fails
END_VAR
VAR_INST
	_inst_arrParams: T_ApiParameterList; // Parameters array
	_inst_arrOutputs: T_ApiParameterList; // Outputs array
	_inst_strRet: T_ApiParamValue; // Return string from the router
	_inst_intStep: INT; // Current method step
	_inst_fbParams: FB_ApiParamBuilder; // Parameter builder FB
END_VAR
VAR
	_bComplete: BOOL; // True if the routing finishes
	_intRet: INT; // Return string converted to an integer
	_bResult : BOOL; // Output of the method
	_pArgs: PVOID; // Arguments pointer
END_VAR
_bResult := FALSE;

// Recover from premature stop
bResetBusy := TRUE;
_inst_intStep := intResetStep;

// Steps
CASE _inst_intStep OF
	0: // Wait for no error and router not busy
		IF (NOT THIS^.P_bError) AND (NOT bRouterBusy) AND THIS^.P_bConnected THEN
			bRouterBusy := TRUE;
			_inst_intStep := _inst_intStep + 10;
		ELSIF (NOT THIS^.P_bError) AND (NOT THIS^.P_bConnected) THEN
			_bResult := TRUE;
		END_IF
		
	10: // Initialize parameters
		THIS^.M_LogMessage(_strSTART_MSG);
		_inst_fbParams.M_ClearParameters();
		_pArgs := _inst_fbParams.M_AddEmptyStruct('args');
		_inst_fbParams.M_OutputToParameterList(_inst_arrParams);
		_inst_intStep := _inst_intStep + 10;
		
	20: // Route the command
		_bComplete := M_RouterHelper(
			_in_strMethodName := _strCOMMAND_NAME, 
			_in_timeTimeout := _timeCOMMAND_TIMEOUT,
			_inout_arrParams := _inst_arrParams,
			_inout_arrOutputs := _inst_arrOutputs,
			_out_strReturnValue=>_inst_strRet);
		
		// If route completed, move to next step
		IF _bComplete THEN
			_inst_intStep := _inst_intStep + 10;
			bRouterBusy := FALSE;
		ELSIF THIS^.P_bError THEN
			_inst_intStep := 0;
			bRouterBusy := FALSE;
		END_IF
		
	30: // Parse results
		_intRet := STRING_TO_INT(_inst_strRet);
		IF _intRet >= 0 THEN
			_bResult := TRUE;
			THIS^.M_LogMessage(_strEND_MSG);
			_inst_fbParams.M_LoadFromParameterList(_inst_arrOutputs);
			bConnected := TRUE;
			
		// Set error if command failed
		ELSE
			THIS^.M_SetError(_udintERROR_ID, _strERROR_MSG);
		END_IF
		
		// Go back to start
		_inst_intStep := 0;
END_CASE

M_Reset := _bResult;
intResetStep := _inst_intStep;
END_METHOD

(* This property should be TRUE while any method in this interface is actively
	executing, or FALSE otherwise. *)
PROPERTY P_bResetBusy : BOOL
GET
P_bResetBusy := bResetBusy;
END_GET
END_PROPERTY

(* This method is a template for any methods that use the API. *)
METHOD M_Trigger : BOOL
VAR CONSTANT
	_strCOMMAND_NAME : T_MaxString	:= 'Trigger'; // Name of the API method
	_timeCOMMAND_TIMEOUT : TIME		:= T#30S; // Max time to receive API response
	_strSTART_MSG : T_MaxString		:= 'Triggering...'; // Prints when method starts
	_strEND_MSG : T_MaxString		:= 'Trigger complete.'; // Prints when method finishes
	_udintERROR_ID : UDINT			:= E_ApiDeviceError.CommandFault; // Error ID to set if command fails
	_strERROR_MSG : T_MaxString		:= 'Triggering failed!'; // Error message to set if command fails
END_VAR
VAR_INST
	_inst_arrParams: T_ApiParameterList; // Parameters array
	_inst_arrOutputs: T_ApiParameterList; // Outputs array
	_inst_strRet: T_ApiParamValue; // Return string from the router
	_inst_intStep: INT; // Current method step
	_inst_fbParams: FB_ApiParamBuilder; // Parameter builder FB
END_VAR
VAR
	_bComplete: BOOL; // True if the routing finishes
	_intRet: INT; // Return string converted to an integer
	_bResult : BOOL; // Output of the method
	_pArgs: PVOID; // Arguments pointer
END_VAR
_bResult := FALSE;

// Recover from premature stop
bTriggerBusy := TRUE;
_inst_intStep := intTriggerStep;

// Steps
CASE _inst_intStep OF
	0: // Wait for no error and router not busy
		IF NOT THIS^.P_bError AND NOT bRouterBusy THEN
			bRouterBusy := TRUE;
			_inst_intStep := _inst_intStep + 10;
		END_IF
		
	10: // Initialize parameters
		THIS^.M_LogMessage(_strSTART_MSG);
		_inst_fbParams.M_ClearParameters();
		_pArgs := _inst_fbParams.M_AddEmptyStruct('args');
		_inst_fbParams.M_AddStructMember(_pArgs, 'filename', in_strProgramName);
		_inst_fbParams.M_AddStructMember(_pArgs, 'guide', in_bGuide);
		_inst_fbParams.M_AddStructMember(_pArgs, 'dryrun', in_bDryrun);
		_inst_fbParams.M_AddStructMember(_pArgs, 'savefile', in_bSaveFile);
		_inst_fbParams.M_AddStructMember(_pArgs, 'signalMonitorOff', in_bSignalMonitorOff);
		_inst_fbParams.M_AddStructMember(_pArgs, 'signalMonitorOn', in_bSignalMonitorOn);
		_inst_fbParams.M_AddStructMember(_pArgs, 'group', in_strGroup);
		_inst_fbParams.M_OutputToParameterList(_inst_arrParams);
		_inst_intStep := _inst_intStep + 10;
		
	20: // Route the command
		_bComplete := M_RouterHelper(
			_in_strMethodName := _strCOMMAND_NAME, 
			_in_timeTimeout := _timeCOMMAND_TIMEOUT,
			_inout_arrParams := _inst_arrParams,
			_inout_arrOutputs := _inst_arrOutputs,
			_out_strReturnValue=>_inst_strRet);
		
		// If route completed, move to next step
		IF _bComplete THEN
			_inst_intStep := _inst_intStep + 10;
			bRouterBusy := FALSE;
		ELSIF THIS^.P_bError THEN
			_inst_intStep := 0;
			bRouterBusy := FALSE;
		END_IF
		
	30: // Parse results
		_intRet := STRING_TO_INT(_inst_strRet);
		IF _intRet > 0 THEN
			_bResult := TRUE;
			THIS^.M_LogMessage(_strEND_MSG);
			_inst_fbParams.M_LoadFromParameterList(_inst_arrOutputs);
			
		// Set error if command failed
		ELSE
			THIS^.M_SetError(_udintERROR_ID, _strERROR_MSG);
		END_IF
		
		// Go back to start
		_inst_intStep := 0;
END_CASE

M_Trigger := _bResult;
intTriggerStep := _inst_intStep;
END_METHOD

ACTION A_CommandRecovery:
(*
	Tell methods to reset if they were not called in the last cycle.
	Make sure to call A_CommandRecovery in function block body.
*)

(*	TEMPLATE: Copy and replace busy/reset variables with busy/reset
	variables of relevant method. *)
IF NOT bTemplateBusy AND intTemplateStep > 0 THEN
	intTemplateStep := 0;
	bRouterBusy := FALSE;
	THIS^.M_LogWarning('M_CommandTemplate ended prematurely!');
END_IF
bTemplateBusy := FALSE;

IF NOT bConnectBusy AND intConnectStep > 0 THEN
	intConnectStep := 0;
	bRouterBusy := FALSE;
	THIS^.M_LogWarning('M_Connect ended prematurely!');
END_IF
bConnectBusy := FALSE;

IF NOT bDisconnectBusy AND intDisconnectStep > 0 THEN
	intDisconnectStep := 0;
	bRouterBusy := FALSE;
	THIS^.M_LogWarning('M_Disconnect ended prematurely!');
END_IF
bDisconnectBusy := FALSE;

IF NOT bGetConnectStatusBusy AND intGetConnectStatusStep > 0 THEN
	intGetConnectStatusStep := 0;
	bRouterBusy := FALSE;
	THIS^.M_LogWarning('M_GetConnectStatus ended prematurely!');
END_IF
bGetConnectStatusBusy := FALSE;

IF NOT bEnableBusy AND intEnableStep > 0 THEN
	intEnableStep := 0;
	bRouterBusy := FALSE;
	THIS^.M_LogWarning('M_Enable ended prematurely!');
END_IF
bEnableBusy := FALSE;

IF NOT bDisableBusy AND intDisableStep > 0 THEN
	intDisableStep := 0;
	bRouterBusy := FALSE;
	THIS^.M_LogWarning('M_Disable ended prematurely!');
END_IF
bDisableBusy := FALSE;

IF NOT bGetEnableStatusBusy AND intGetEnableStatusStep > 0 THEN
	intGetEnableStatusStep := 0;
	bRouterBusy := FALSE;
	THIS^.M_LogWarning('M_GetEnableStatus ended prematurely!');
END_IF
bGetEnableStatusBusy := FALSE;

IF NOT bPowerOnBusy AND intPowerOnStep > 0 THEN
	intPowerOnStep := 0;
	bRouterBusy := FALSE;
	THIS^.M_LogWarning('M_PowerOn ended prematurely!');
END_IF
bPowerOnBusy := FALSE;

IF NOT bPowerOffBusy AND intPowerOffStep > 0 THEN
	intPowerOffStep := 0;
	bRouterBusy := FALSE;
	THIS^.M_LogWarning('M_PowerOff ended prematurely!');
END_IF
bPowerOffBusy := FALSE;

IF NOT bGetPowerStatusBusy AND intGetPowerStatusStep > 0 THEN
	intGetPowerStatusStep := 0;
	bRouterBusy := FALSE;
	THIS^.M_LogWarning('M_GetPowerStatus ended prematurely!');
END_IF
bGetPowerStatusBusy := FALSE;

IF NOT bGetCurrentProgramBusy AND intGetCurrentProgramStep > 0 THEN
	intGetCurrentProgramStep := 0;
	bRouterBusy := FALSE;
	THIS^.M_LogWarning('M_GetCurrentProgram ended prematurely!');
END_IF
bGetCurrentProgramBusy := FALSE;

IF NOT bGetProgramStateBusy AND intGetProgramStateStep > 0 THEN
	intGetProgramStateStep := 0;
	bRouterBusy := FALSE;
	THIS^.M_LogWarning('M_GetProgramState ended prematurely!');
END_IF
bGetProgramStateBusy := FALSE;

IF NOT bLoadProgramBusy AND intLoadProgramStep > 0 THEN
	intLoadProgramStep := 0;
	bRouterBusy := FALSE;
	THIS^.M_LogWarning('M_LoadProgram ended prematurely!');
END_IF
bLoadProgramBusy := FALSE;

IF NOT bPauseProgramBusy AND intPauseProgramStep > 0 THEN
	intPauseProgramStep := 0;
	bRouterBusy := FALSE;
	THIS^.M_LogWarning('M_PauseProgram ended prematurely!');
END_IF
bPauseProgramBusy := FALSE;

IF NOT bStartProgramBusy AND intStartProgramStep > 0 THEN
	intStartProgramStep := 0;
	bRouterBusy := FALSE;
	THIS^.M_LogWarning('M_StartProgram ended prematurely!');
END_IF
bStartProgramBusy := FALSE;

IF NOT bStopProgramBusy AND intStopProgramStep > 0 THEN
	intStopProgramStep := 0;
	bRouterBusy := FALSE;
	THIS^.M_LogWarning('M_StopProgram ended prematurely!');
END_IF
bStopProgramBusy := FALSE;

IF NOT bResetBusy AND intResetStep > 0 THEN
	intResetStep := 0;
	bRouterBusy := FALSE;
	THIS^.M_LogWarning('M_ResetBusy ended prematurely!');
END_IF
bResetBusy := FALSE;

IF NOT bAbortBusy AND intAbortStep > 0 THEN
	intAbortStep := 0;
	bRouterBusy := FALSE;
	THIS^.M_LogWarning('M_Abort ended prematurely!');
END_IF
bAbortBusy := FALSE;

IF NOT bTriggerBusy AND intTriggerStep > 0 THEN
	intTriggerStep := 0;
	bRouterBusy := FALSE;
	THIS^.M_LogWarning('M_CommandTemplate ended prematurely!');
END_IF
bTriggerBusy := FALSE;

IF NOT bRouterHelperBusy AND intRouterHelperStep > 0 THEN
	intRouterHelperStep := 0;
	bRouterBusy := FALSE;
	THIS^.M_LogWarning('M_RouterHelper ended prematurely!');
END_IF
bRouterHelperBusy := FALSE;
END_ACTION

(* This method is a template for any methods that use the API. *)
METHOD PRIVATE M_CommandTemplate : BOOL
VAR CONSTANT
	_strCOMMAND_NAME : T_MaxString	:= 'CommandTemplate'; // Name of the API method
	_timeCOMMAND_TIMEOUT : TIME		:= T#30S; // Max time to receive API response
	_strSTART_MSG : T_MaxString		:= 'Routing command...'; // Prints when method starts
	_strEND_MSG : T_MaxString		:= 'Command complete.'; // Prints when method finishes
	_udintERROR_ID : UDINT			:= E_ApiDeviceError.CommandFault; // Error ID to set if command fails
	_strERROR_MSG : T_MaxString		:= 'Command failed!'; // Error message to set if command fails
END_VAR
VAR_INST
	_inst_arrParams: T_ApiParameterList; // Parameters array
	_inst_arrOutputs: T_ApiParameterList; // Outputs array
	_inst_strRet: T_ApiParamValue; // Return string from the router
	_inst_intStep: INT; // Current method step
	_inst_fbParams: FB_ApiParamBuilder; // Parameter builder FB
END_VAR
VAR
	_bComplete: BOOL; // True if the routing finishes
	_intRet: INT; // Return string converted to an integer
	_bResult : BOOL; // Output of the method
	_pArgs: PVOID; // Arguments pointer
END_VAR
_bResult := FALSE;

// Recover from premature stop
(* TEMPLATE: Replace bTemplateBusy and intTemplateStep with relevant
	variables for specific command. Also replace M_CommandTemplate
	and intTemplateStep in the last two lines of this method. *)
bTemplateBusy := TRUE;
_inst_intStep := intTemplateStep;

// Steps
(* TEMPLATE: Parameters should be added in step 10, and output
	parsing should be added in step 30. *)
CASE _inst_intStep OF
	0: // Wait for no error and router not busy
		IF NOT THIS^.P_bError AND NOT bRouterBusy THEN
			bRouterBusy := TRUE;
			_inst_intStep := _inst_intStep + 10;
		END_IF
		
	10: // Initialize parameters
		THIS^.M_LogMessage(_strSTART_MSG);
		_inst_fbParams.M_ClearParameters();
		_pArgs := _inst_fbParams.M_AddEmptyStruct('args');
		// TEMPLATE: Add any parameters here
		_inst_fbParams.M_OutputToParameterList(_inst_arrParams);
		_inst_intStep := _inst_intStep + 10;
		
	20: // Route the command
		_bComplete := M_RouterHelper(
			_in_strMethodName := _strCOMMAND_NAME, 
			_in_timeTimeout := _timeCOMMAND_TIMEOUT,
			_inout_arrParams := _inst_arrParams,
			_inout_arrOutputs := _inst_arrOutputs,
			_out_strReturnValue=>_inst_strRet);
		
		// If route completed, move to next step
		IF _bComplete THEN
			_inst_intStep := _inst_intStep + 10;
			bRouterBusy := FALSE;
		ELSIF THIS^.P_bError THEN
			_inst_intStep := 0;
			bRouterBusy := FALSE;
		END_IF
		
	30: // Parse results
		_intRet := STRING_TO_INT(_inst_strRet);
		IF _intRet > 0 THEN
			_bResult := TRUE;
			THIS^.M_LogMessage(_strEND_MSG);
			_inst_fbParams.M_LoadFromParameterList(_inst_arrOutputs);
			// TEMPLATE: Do any parsing here
			
		// Set error if command failed
		ELSE
			THIS^.M_SetError(_udintERROR_ID, _strERROR_MSG);
		END_IF
		
		// Go back to start
		_inst_intStep := 0;
END_CASE
// TEMPLATE: Replace with method name and step variable
M_CommandTemplate := _bResult;
intTemplateStep := _inst_intStep;
END_METHOD

(*
Sends the given method to the API and receives and partially parses the result.
*)
METHOD PRIVATE M_RouterHelper : BOOL
VAR_INPUT
	(* Name of the method to call. *)
	_in_strMethodName : T_MaxString;
	(* Maximum time to wait for method response. *)
	_in_timeTimeout : TIME;
END_VAR
VAR_IN_OUT
	(* The array of parameters to send to the API. *)
	_inout_arrParams : T_ApiParameterList;
	(* The array that gets populated with any method output data. *)
	_inout_arrOutputs : T_ApiParameterList;
END_VAR
VAR_OUTPUT
	(* JSON string of the method return value. *)
	_out_strReturnValue: T_ApiParamValue;
END_VAR
VAR_INST
	(* Current step. *)
	_inst_intStep: INT;
	(* True if the method executed. *)
	_inst_bExec: BOOL;
	(* Return string of the method. *)
	_inst_strRet: T_ApiParamValue;
END_VAR
VAR
	(* True once the command routing finishes. *)
	_bComplete: BOOL;
	(* True once the API connects. *)
	_bApiConnect: BOOL;
END_VAR
// Recover from premature stop
bRouterHelperBusy := TRUE;
_inst_intStep := intRouterHelperStep;

// Steps
CASE _inst_intStep OF
	0: // Start process only if there is no error on this FB
		IF NOT THIS^.P_bError THEN
			in_fbApi.M_ClearError();
			_inst_intStep := 10;
		END_IF
		
	10: // Check if command router is connected
		IF NOT in_fbApi.P_bConnected THEN
			_inst_intStep := 20; // Go to API connect step
		ELSE
			_inst_intStep := 30; // Go to route command step
		END_IF
		
	20: // Connect to the command router
		_bApiConnect := in_fbApi.M_Connect();
		IF _bApiConnect THEN
			_inst_intStep := _inst_intStep + 10; // Go to next step
		ELSIF in_fbApi.P_bError THEN
			THIS^.M_SetError(E_ApiDeviceError.CommandRouterError, 'Error on command router function block while connecting!');
			_inst_intStep := 0; // Go back to start
		END_IF
		
	30:	// Route the command
		_bComplete := in_fbApi.M_RouteCommand(
			_in_strModuleId := in_strApiModuleId,
			_in_strMethodName := _in_strMethodName,
			_in_timeTimeout := _in_timeTimeout,
			_inout_arrParameters := _inout_arrParams,
			_inout_arrOutputs := _inout_arrOutputs,
			_out_bCommandExecuted => _inst_bExec,
			_out_strReturnValue => _inst_strRet);
		IF _bComplete THEN
			_inst_intStep := _inst_intStep + 10; // Go to next step
		ELSIF in_fbApi.P_bError THEN
			THIS^.M_SetError(E_ApiDeviceError.CommandRouterError, 'Error on command router function block while routing command!');
			_inst_intStep := 0; // Go back to start
		END_IF
		
	40: // Check result then go back to start
		IF NOT _inst_bExec THEN
			THIS^.M_SetError(E_ApiDeviceError.CommandFault, 'Method in API failed to execute!');
		ELSE
			_out_strReturnValue := _inst_strRet;
			M_RouterHelper := TRUE;
		END_IF
		_inst_intStep := 0; // Go back to start
END_CASE

intRouterHelperStep := _inst_intStep;
END_METHOD

END_FUNCTION_BLOCK

// Concrete/Keyence MDX-2000/FB_KeyenceLaserMarkerMDX2000
FUNCTION_BLOCK PUBLIC FB_KeyenceLaserMarkerMDX2000 EXTENDS FB_LaserMarker
	IMPLEMENTS 
		I_Connectable,
		I_Resettable,
		I_Programmable,
		I_Markable
VAR_INPUT
	in_fbApi : REFERENCE TO FB_CommandRouter; (* Device API connection to the "". *)
	// Marking program name
	in_strProgram	: Sensata_Common.T_MaxString;	
//Send Marking Parameters Block Range
//	in_PartNoStart : INT;
//	in_PartNoEnd : INT;
//	in_BlockRangeData : T_MaxString;
END_VAR
VAR_OUTPUT
END_VAR
VAR
	// Connectable
	bApiConnected: BOOL; (* TRUE if the API is connected. *) // 
	bConnected: BOOL; (* TRUE if the Laser is connected. *)
	bConnecting: BOOL; (* TRUE while the connect command is running. *)
	bDisconnecting: BOOL; (* TRUE while the disconnect command is running. *)
	bActive: BOOL;
   	bSendingSendLaserProgram : BOOL;
	bEnabled : BOOL; // Value of P_bEnabled
	enumProgramState: E_PROGRAMSTATE; // Value of P_enumProgramState
	bRouterBusy: BOOL; // TRUE while M_RouterHelper is being used by a method
	bResetBusy: BOOL; // Value of P_bResetBusy
	bPoweredOn: BOOL; // Value of P_bPoweredOn
	strLoadedProgram: STRING(255); // Value of P_strLoadedProgram
	
	//Variables added to recover easily in a particular step number after abort.

	//Command Busy bits
	bRouterHelperBusy: BOOL;
	bMConnectBusy : BOOL;
	bMDisconnectBusy : BOOL;
	bMGetConnectStatusBusy : BOOL;
	bMPeakCurrentProgramBusy : BOOL;
	bMSendMarkingParamsBusy : BOOL;
	bMStartMarkingBusy : BOOL;
	bMStopMarkingBusy : BOOL;
	bMUpdateAllMarkingInfoBusy : BOOL;
	bMUpdateSingleBlockInfoBusy : BOOL;
	bMGetCurrentProgBusy : BOOL;
	bMLoadProgramBusy : BOOL;
	bMSaveCurrentLaserProgramtoPCBusy : BOOL;
	bMSendProgramToLaserBusy :BOOL;
	bMStartProgramBusy : BOOL;
	bMUpdateSingleProgramBlockDataBusy : BOOL;
	bMUpdateSingleProgramBlockMarkingEnabledBusy : BOOL;
	bMGetLaserActivatedStatusBusy : BOOL;
	bMGetLaserErrorStatusBusy : BOOL;
	bMGetLaserMarkingStatusBusy : BOOL;
	bMGetLaserStatusBusy : BOOL;
	bMClearErrorBusy : BOOL;
	bMResetBusy : BOOL;
	
	//Command Steps
	intRouterHelperStep: INT;
	intMConnectStep : INT;
	intMDisconnectStep : INT;
	intMGetConnectStatusStep : INT;
	intMPeakCurrentProgramStep : INT;
	intMSendMarkingParamsStep : INT;
	intMStartMarkingStep : INT;
	intMStopMarkingStep : INT;
	intMUpdateAllMarkingInfoStep : INT;
	intMUpdateSingleBlockInfoStep : INT;
	intMGetCurrentProgStep : INT;
	intMLoadProgramStep : INT;
	intMSaveCurrentLaserProgramtoPC : INT;
	intMSendProgramToLaserStep :INT;
	intMStartProgramStep : INT;
	intMUpdateSingleProgramBlockDataStep : INT;
	intMUpdateSingleProgramBlockMarkingEnabledStep : INT;
	intMGetLaserActivatedStatusStep : INT;
	intMGetLaserErrorStatusStep : INT;
	intMGetLaserMarkingStatusStep : INT;
	intMGetLaserStatusStep : INT;
	intMClearErrorStep : INT;
	intMResetStep : INT;
	
END_VAR

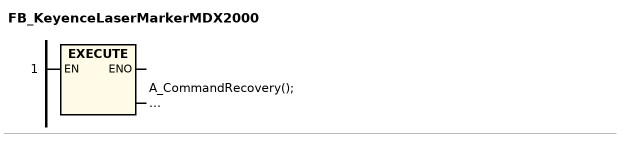
// NETWORK 1
A_CommandRecovery();

METHOD M_Connect : BOOL
VAR_INPUT
	
END_VAR

VAR_OUTPUT
	
END_VAR

VAR CONSTANT
	_strCOMMAND_NAME : T_MaxString	:= 'Connect'; // Name of the API method
	_timeCOMMAND_TIMEOUT : TIME		:= T#30S; // Max time to receive API response
	_strSTART_MSG : T_MaxString		:= 'Connecting'; // Prints when method starts
	_strEND_MSG : T_MaxString		:= 'Connected'; // Prints when method finishes
	_udintERROR_ID : UDINT			:= KeyenceLaserMarkerMDX2000_Error.FailedToConnect; // Error ID to set if command fails
	_strERROR_MSG : T_MaxString		:= 'Failed to connect to Laser Marker!'; // Error message to set if command fails
END_VAR

VAR_INST
	_inst_arrParams: T_ApiParameterList; // Parameters array
	_inst_arrOutputs: T_ApiParameterList; // Outputs array
	_inst_strRet: T_ApiParamValue; // Return string from the router
	_inst_intStep: INT; // Current method step
	_inst_fbParams: FB_ApiParamBuilder; // Parameter builder FB
END_VAR

VAR
	
	_bComplete: BOOL; // True if the routing finishes
	_intRet: INT; // Return string converted to an integer
	_bResult : BOOL; // Output of the method

END_VAR
_bResult := FALSE;
_inst_intStep := intMConnectStep;
bMConnectBusy := TRUE;
//END_IF
CASE _inst_intStep OF
	0: // Wait for no error and router not busy
		IF NOT THIS^.P_bError AND NOT bRouterBusy THEN
			bRouterBusy := TRUE;
			_inst_intStep := _inst_intStep + 10;
		END_IF
		
	10: // Initialize parameters
		THIS^.M_LogMessage(_strSTART_MSG);
		_inst_fbParams.M_ClearParameters();
		// ADD ANY PARAMETERS HERE
		_inst_fbParams.M_OutputToParameterList(_inst_arrParams);
		_inst_intStep := _inst_intStep + 10;
		
	20: // Route the command
		_bComplete := M_RouterHelper(
			_in_strMethodName := _strCOMMAND_NAME, 
			_in_timeTimeout := _timeCOMMAND_TIMEOUT,
			_inout_arrParams := _inst_arrParams,
			_inout_arrOutputs := _inst_arrOutputs,
			_out_strReturnValue=>_inst_strRet);
		
		// If route completed, move to next step
		IF _bComplete THEN
			_inst_intStep := _inst_intStep + 10;
			bRouterBusy := FALSE;
		ELSIF THIS^.P_bError THEN
			_inst_intStep := 0;
			bRouterBusy := FALSE;
		END_IF
		
	30: // Parse results
		_intRet := STRING_TO_INT(_inst_strRet);
		IF _intRet > 0 THEN
			_bResult := TRUE;
			THIS^.M_LogMessage(_strEND_MSG);
			// DO ANY PARSING HERE
			bConnected := TRUE;
		// Set error if command failed
		ELSE
			THIS^.M_SetError(_udintERROR_ID, _strERROR_MSG);
		END_IF
		// Go back to start
		_inst_intStep := 0;
END_CASE
M_Connect := _bResult;
intMConnectStep := _inst_intStep;
END_METHOD

METHOD PUBLIC M_Disconnect : BOOL

VAR CONSTANT
	_strCOMMAND_NAME : T_MaxString	:= 'Disconnect'; // Name of the API method
	_timeCOMMAND_TIMEOUT : TIME		:= T#30S; // Max time to receive API response
	_strSTART_MSG : T_MaxString		:= 'Disconnecting'; // Prints when method starts
	_strEND_MSG : T_MaxString		:= 'Disconnected'; // Prints when method finishes
	_udintERROR_ID : UDINT			:= KeyenceLaserMarkerMDX2000_Error.FailedToDisconnect; // Error ID to set if command fails
	_strERROR_MSG : T_MaxString		:= 'Failed to Disconnect from Laser Marker!'; // Error message to set if command fails
END_VAR

VAR_INST
	_inst_arrParams: T_ApiParameterList; // Parameters array
	_inst_arrOutputs: T_ApiParameterList; // Outputs array
	_inst_strRet: T_ApiParamValue; // Return string from the router
	_inst_intStep: INT; // Current method step
	_inst_fbParams: FB_ApiParamBuilder; // Parameter builder FB
END_VAR

VAR
	_bComplete: BOOL; // True if the routing finishes
	_intRet: INT; // Return string converted to an integer
	_bResult : BOOL; // Output of the method
END_VAR
_bResult := FALSE;
bMDisconnectBusy := TRUE;
_inst_intStep := intMDisconnectStep;
CASE _inst_intStep OF
	0: // Wait for no error and router not busy
		IF NOT THIS^.P_bError AND NOT bRouterBusy THEN
			bRouterBusy := TRUE;
			_inst_intStep := _inst_intStep + 10;
		END_IF
		
	10: // Initialize parameters
		THIS^.M_LogMessage(_strSTART_MSG);
		_inst_fbParams.M_ClearParameters();
		// ADD ANY PARAMETERS HERE
		_inst_fbParams.M_OutputToParameterList(_inst_arrParams);
		_inst_intStep := _inst_intStep + 10;
		
	20: // Route the command
		_bComplete := M_RouterHelper(
			_in_strMethodName := _strCOMMAND_NAME, 
			_in_timeTimeout := _timeCOMMAND_TIMEOUT,
			_inout_arrParams := _inst_arrParams,
			_inout_arrOutputs := _inst_arrOutputs,
			_out_strReturnValue=>_inst_strRet);
		
		// If route completed, move to next step
		IF _bComplete THEN
			_inst_intStep := _inst_intStep + 10;
			bRouterBusy := FALSE;
		ELSIF THIS^.P_bError THEN
			_inst_intStep := 0;
			bRouterBusy := FALSE;
		END_IF
		
	30: // Parse results
		_intRet := STRING_TO_INT(_inst_strRet);
		IF _intRet > 0 THEN
			_bResult := TRUE;
			THIS^.M_LogMessage(_strEND_MSG);
			// DO ANY PARSING HERE
			bConnected := TRUE;
//			P_bConnected := FALSE;
		// Set error if command failed
		ELSE
			THIS^.M_SetError(_udintERROR_ID, _strERROR_MSG);
		END_IF
		// Go back to start
		_inst_intStep := 0;
END_CASE
M_Disconnect := _bResult;
intMDisconnectStep := _inst_intStep;
END_METHOD

(* This method should explicitly check the connection status of the device.
	Once the connection status is known, this method should return TRUE.
	If this method fails, P_bConnected should be set to FALSE since the device
	is not absolutely known to still be connected. *)
METHOD M_GetConnectStatus : BOOL
VAR_OUTPUT
	(* This should return TRUE if all connections required to make the device
		function properly are known to be connected, and FALSE otherwise. *)
	bConnected	: BOOL;
END_VAR
VAR CONSTANT
	_strCOMMAND_NAME : T_MaxString	:= 'GetConnectionStatus'; // Name of the API method
	_timeCOMMAND_TIMEOUT : TIME		:= T#30S; // Max time to receive API response
	_strSTART_MSG : T_MaxString		:= 'GettingConnectionStatus'; // Prints when method starts
	_strEND_MSG : T_MaxString		:= 'GotConnectionStatus'; // Prints when method finishes
	_udintERROR_ID : UDINT			:= KeyenceLaserMarkerMDX2000_Error.FailedToGetConnectStatus; // Error ID to set if command fails
	_strERROR_MSG : T_MaxString		:= 'Failed to Get Connection Status from Laser Marker!'; // Error message to set if command fails
END_VAR

VAR_INST
	_inst_arrParams: T_ApiParameterList; // Parameters array
	_inst_arrOutputs: T_ApiParameterList; // Outputs array
	_inst_strRet: T_ApiParamValue; // Return string from the router
	_inst_intStep: INT; // Current method step
	_inst_fbParams: FB_ApiParamBuilder; // Parameter builder FB
END_VAR

VAR
	
	_bComplete: BOOL; // True if the routing finishes
	_intRet: INT; // Return string converted to an integer
	_bResult : BOOL; // Output of the method

END_VAR
bConnected := P_bConnected;
bMGetConnectStatusBusy := TRUE;
_inst_intStep := intMGetConnectStatusStep;
_bResult := FALSE;
//bCommandBusy := TRUE;
//IF bResetCommands THEN
//	_inst_intStep := 0;
//END_IF
CASE _inst_intStep OF
	0: // Wait for no error and router not busy
		IF NOT THIS^.P_bError AND NOT bRouterBusy THEN
			bRouterBusy := TRUE;
			_inst_intStep := _inst_intStep + 10;
		END_IF
		
	10: // Initialize parameters
		THIS^.M_LogMessage(_strSTART_MSG);
		_inst_fbParams.M_ClearParameters();
		// ADD ANY PARAMETERS HERE
		_inst_fbParams.M_OutputToParameterList(_inst_arrParams);
		_inst_intStep := _inst_intStep + 10;
		
	20: // Route the command
		_bComplete := M_RouterHelper(
			_in_strMethodName := _strCOMMAND_NAME, 
			_in_timeTimeout := _timeCOMMAND_TIMEOUT,
			_inout_arrParams := _inst_arrParams,
			_inout_arrOutputs := _inst_arrOutputs,
			_out_strReturnValue=>_inst_strRet);
		
		// If route completed, move to next step
		IF _bComplete THEN
			_inst_intStep := _inst_intStep + 10;
			bRouterBusy := FALSE;
		ELSIF THIS^.P_bError THEN
			_inst_intStep := 0;
			bRouterBusy := FALSE;
		END_IF
		
	30: // Parse results
		_intRet := STRING_TO_INT(_inst_strRet);
		IF _intRet > 0 THEN
			_bResult := TRUE;
			THIS^.M_LogMessage(_strEND_MSG);
			// DO ANY PARSING HERE
			_inst_fbParams.M_LoadFromParameterList(_inst_arrOutputs);
			bConnected := _inst_fbParams.M_ParseBool(_inst_fbParams.M_GetParameter('connected'));
//			P_bConnected := TRUE;
		// Set error if command failed
		ELSE
			THIS^.M_SetError(_udintERROR_ID, _strERROR_MSG);
		END_IF
		// Go back to start
		_inst_intStep := 0;
END_CASE

M_GetConnectStatus := _bResult;
intMGetConnectStatusStep := _inst_intStep;
END_METHOD

(* This property should be TRUE while any method in this interface is actively
	executing, or FALSE otherwise. *)
PROPERTY P_bConnectBusy : BOOL
GET
P_bConnectBusy := bConnecting OR bDisconnecting;
END_GET
END_PROPERTY

(* This should be set to TRUE if M_Connect is successful or M_GetConnectStatus
	determines the device to be connected, and set to FALSE if M_Disconnect is
	called at all, M_GetConnectStatus fails, or M_GetConnectStatus determines
	the device to be not connected. *)
PROPERTY P_bConnected : BOOL
GET
P_bConnected := bApiConnected AND bConnected;
END_GET
END_PROPERTY

METHOD PUBLIC M_PeakCurrentProgram : BOOL
VAR_INPUT
END_VAR

VAR CONSTANT
	_strCOMMAND_NAME : T_MaxString	:= 'PeakCurrentProgram'; // Name of the API method
	_timeCOMMAND_TIMEOUT : TIME		:= T#30S; // Max time to receive API response
	_strSTART_MSG : T_MaxString		:= 'PeakingCurrentProgram'; // Prints when method starts
	_strEND_MSG : T_MaxString		:= 'PeakedCurrentProgram'; // Prints when method finishes
	_udintERROR_ID : UDINT			:= KeyenceLaserMarkerMDX2000_Error.FailedToPeakCurrentProgram; // Error ID to set if command fails
	_strERROR_MSG : T_MaxString		:= 'Failed to Peak Current Program in Laser Marker!'; // Error message to set if command fails
END_VAR

VAR_INST
	_inst_arrParams: T_ApiParameterList; // Parameters array
	_inst_arrOutputs: T_ApiParameterList; // Outputs array
	_inst_strRet: T_ApiParamValue; // Return string from the router
	_inst_intStep: INT; // Current method step
	_inst_fbParams: FB_ApiParamBuilder; // Parameter builder FB
END_VAR

VAR
		
	_bComplete: BOOL; // True if the routing finishes
	_intRet: INT; // Return string converted to an integer
	_bResult : BOOL; // Output of the method
END_VAR
_bResult := FALSE;
_inst_intStep := intMPeakCurrentProgramStep;
bMPeakCurrentProgramBusy := TRUE;
CASE _inst_intStep OF
	0: // Wait for no error and router not busy
		IF NOT THIS^.P_bError AND NOT bRouterBusy THEN
			bRouterBusy := TRUE;
			_inst_intStep := _inst_intStep + 10;
		END_IF
		
	10: // Initialize parameters
		THIS^.M_LogMessage(_strSTART_MSG);
		_inst_fbParams.M_ClearParameters();
		// ADD ANY PARAMETERS HERE
		_inst_fbParams.M_OutputToParameterList(_inst_arrParams);
		_inst_intStep := _inst_intStep + 10;
		
	20: // Route the command
		_bComplete := M_RouterHelper(
			_in_strMethodName := _strCOMMAND_NAME, 
			_in_timeTimeout := _timeCOMMAND_TIMEOUT,
			_inout_arrParams := _inst_arrParams,
			_inout_arrOutputs := _inst_arrOutputs,
			_out_strReturnValue=>_inst_strRet);
		
		// If route completed, move to next step
		IF _bComplete THEN
			_inst_intStep := _inst_intStep + 10;
			bRouterBusy := FALSE;
		ELSIF THIS^.P_bError THEN
			_inst_intStep := 0;
			bRouterBusy := FALSE;
		END_IF
		
	30: // Parse results
		_intRet := STRING_TO_INT(_inst_strRet);
		IF _intRet > 0 THEN
			_bResult := TRUE;
			THIS^.M_LogMessage(_strEND_MSG);
			// DO ANY PARSING HERE
			bConnected := TRUE;
		// Set error if command failed
		ELSE
			THIS^.M_SetError(_udintERROR_ID, _strERROR_MSG);
		END_IF
		// Go back to start
		_inst_intStep := 0;
END_CASE
M_PeakCurrentProgram := _bResult;
intMPeakCurrentProgramStep := _inst_intStep;
END_METHOD

METHOD PUBLIC M_SendMarkingParams_BlockRange : BOOL
VAR_INPUT
	in_MarkEnabled : BOOL;
END_VAR

VAR CONSTANT
	_strCOMMAND_NAME : T_MaxString	:= 'SendMarkingParams_BlockRange'; // Name of the API method
	_timeCOMMAND_TIMEOUT : TIME		:= T#30S; // Max time to receive API response
	_strSTART_MSG : T_MaxString		:= 'SendingMarkingParamsforBlockRange'; // Prints when method starts
	_strEND_MSG : T_MaxString		:= 'SentMarkingParamsforBlockRange'; // Prints when method finishes
	_udintERROR_ID : UDINT			:= KeyenceLaserMarkerMDX2000_Error.FailedToSendMarkingParams_BlockRange; // Error ID to set if command fails
	_strERROR_MSG : T_MaxString		:= 'Failed to send marking params for Block Range!'; // Error message to set if command fails
END_VAR

VAR_INST
	_inst_arrParams: T_ApiParameterList; // Parameters array
	_inst_arrOutputs: T_ApiParameterList; // Outputs array
	_inst_strRet: T_ApiParamValue; // Return string from the router
	_inst_intStep: INT; // Current method step
	_inst_fbParams: FB_ApiParamBuilder; // Parameter builder FB
END_VAR

VAR
	_bComplete: BOOL; // True if the routing finishes
	_intRet: INT; // Return string converted to an integer
	_bResult : BOOL; // Output of the method
END_VAR
_bResult := FALSE;
_inst_intStep := intMSendMarkingParamsStep;
bMSendMarkingParamsBusy := TRUE;
CASE _inst_intStep OF
	0: // Wait for no error and router not busy
		IF NOT THIS^.P_bError AND NOT bRouterBusy THEN
			bRouterBusy := TRUE;
			_inst_intStep := _inst_intStep + 10;
		END_IF
		
	10: // Initialize parameters
		THIS^.M_LogMessage(_strSTART_MSG);
		_inst_fbParams.M_ClearParameters();
		// ADD ANY PARAMETERS HERE
		_inst_fbParams.M_AddParameter('data', in_BlockRangeData);
		_inst_fbParams.M_AddParameter('PartNoStart', in_PartNoStart);
		_inst_fbParams.M_AddParameter('PartNoEnd', in_PartNoEnd);
		_inst_fbParams.M_AddParameter('MarkEnabled', in_MarkEnabled);		
		_inst_fbParams.M_OutputToParameterList(_inst_arrParams);
		_inst_intStep := _inst_intStep + 10;
		
	20: // Route the command
		_bComplete := M_RouterHelper(
			_in_strMethodName := _strCOMMAND_NAME, 
			_in_timeTimeout := _timeCOMMAND_TIMEOUT,
			_inout_arrParams := _inst_arrParams,
			_inout_arrOutputs := _inst_arrOutputs,
			_out_strReturnValue=>_inst_strRet);
		
		// If route completed, move to next step
		IF _bComplete THEN
			_inst_intStep := _inst_intStep + 10;
			bRouterBusy := FALSE;
		ELSIF THIS^.P_bError THEN
			_inst_intStep := 0;
			bRouterBusy := FALSE;
		END_IF
		
	30: // Parse results
		_intRet := STRING_TO_INT(_inst_strRet);
		IF _intRet > 0 THEN
			_bResult := TRUE;
			THIS^.M_LogMessage(_strEND_MSG);
			// DO ANY PARSING HERE
			_inst_fbParams.M_LoadFromParameterList(_inst_arrOutputs);
			bConnected := TRUE;
		// Set error if command failed
		ELSE
			THIS^.M_SetError(_udintERROR_ID, _strERROR_MSG);
		END_IF
		// Go back to start
		_inst_intStep := 0;
END_CASE
M_SendMarkingParams_BlockRange := _bResult;
intMSendMarkingParamsStep := _inst_intStep;
END_METHOD

METHOD PUBLIC M_StartMarking : BOOL
VAR_INPUT
END_VAR

VAR CONSTANT
	_strCOMMAND_NAME : T_MaxString	:= 'StartMarking'; // Name of the API method
	_timeCOMMAND_TIMEOUT : TIME		:= T#30S; // Max time to receive API response
	_strSTART_MSG : T_MaxString		:= 'StartingMarking'; // Prints when method starts
	_strEND_MSG : T_MaxString		:= 'StartedMarking'; // Prints when method finishes
	_udintERROR_ID : UDINT			:= KeyenceLaserMarkerMDX2000_Error.FailedToStartMarking; // Error ID to set if command fails
	_strERROR_MSG : T_MaxString		:= 'Failed to Start Marking by Laser Marker!'; // Error message to set if command fails
END_VAR

VAR_INST
	_inst_arrParams: T_ApiParameterList; // Parameters array
	_inst_arrOutputs: T_ApiParameterList; // Outputs array
	_inst_strRet: T_ApiParamValue; // Return string from the router
	_inst_intStep: INT; // Current method step
	_inst_fbParams: FB_ApiParamBuilder; // Parameter builder FB
END_VAR

VAR
	_bComplete: BOOL; // True if the routing finishes
	_intRet: INT; // Return string converted to an integer
	_bResult : BOOL; // Output of the method
END_VAR
_bResult := FALSE;
bMStartMarkingBusy := TRUE;
_inst_intStep := intMStartMarkingStep;
CASE _inst_intStep OF
	0: // Wait for no error and router not busy
		IF NOT THIS^.P_bError AND NOT bRouterBusy THEN
			bRouterBusy := TRUE;
			_inst_intStep := _inst_intStep + 10;
		END_IF
		
	10: // Initialize parameters
		THIS^.M_LogMessage(_strSTART_MSG);
		_inst_fbParams.M_ClearParameters();
		// ADD ANY PARAMETERS HERE
		_inst_fbParams.M_OutputToParameterList(_inst_arrParams);
		_inst_intStep := _inst_intStep + 10;
		
	20: // Route the command
		_bComplete := M_RouterHelper(
			_in_strMethodName := _strCOMMAND_NAME, 
			_in_timeTimeout := _timeCOMMAND_TIMEOUT,
			_inout_arrParams := _inst_arrParams,
			_inout_arrOutputs := _inst_arrOutputs,
			_out_strReturnValue=>_inst_strRet);
		
		// If route completed, move to next step
		IF _bComplete THEN
			_inst_intStep := _inst_intStep + 10;
			bRouterBusy := FALSE;
		ELSIF THIS^.P_bError THEN
			_inst_intStep := 0;
			bRouterBusy := FALSE;
		END_IF
		
	30: // Parse results
		_intRet := STRING_TO_INT(_inst_strRet);
		IF _intRet > 0 THEN
			_bResult := TRUE;
			THIS^.M_LogMessage(_strEND_MSG);
			// DO ANY PARSING HERE
			bConnected := TRUE;
		// Set error if command failed
		ELSE
			THIS^.M_SetError(_udintERROR_ID, _strERROR_MSG);
		END_IF
		// Go back to start
		_inst_intStep := 0;
END_CASE
M_StartMarking := _bResult;
intMStartMarkingStep := _inst_intStep;
END_METHOD

METHOD PUBLIC M_StopMarking : BOOL
VAR_INPUT
END_VAR

VAR CONSTANT
	_strCOMMAND_NAME : T_MaxString	:= 'StopMarking'; // Name of the API method
	_timeCOMMAND_TIMEOUT : TIME		:= T#30S; // Max time to receive API response
	_strSTART_MSG : T_MaxString		:= 'StoppingMarking'; // Prints when method starts
	_strEND_MSG : T_MaxString		:= 'StoppedMarking'; // Prints when method finishes
	_udintERROR_ID : UDINT			:= KeyenceLaserMarkerMDX2000_Error.FailedToStopMarking; // Error ID to set if command fails
	_strERROR_MSG : T_MaxString		:= 'Failed to Stop Marking by Laser Marker!'; // Error message to set if command fails
END_VAR

VAR_INST
	_inst_arrParams: T_ApiParameterList; // Parameters array
	_inst_arrOutputs: T_ApiParameterList; // Outputs array
	_inst_strRet: T_ApiParamValue; // Return string from the router
	_inst_intStep: INT; // Current method step
	_inst_fbParams: FB_ApiParamBuilder; // Parameter builder FB
END_VAR

VAR
	_bComplete: BOOL; // True if the routing finishes
	_intRet: INT; // Return string converted to an integer
	_bResult : BOOL; // Output of the method
END_VAR
_bResult := FALSE;
bMStopMarkingBusy := TRUE;
_inst_intStep := intMStopMarkingStep;
CASE _inst_intStep OF
	0: // Wait for no error and router not busy
		IF NOT THIS^.P_bError AND NOT bRouterBusy THEN
			bRouterBusy := TRUE;
			_inst_intStep := _inst_intStep + 10;
		END_IF
		
	10: // Initialize parameters
		THIS^.M_LogMessage(_strSTART_MSG);
		_inst_fbParams.M_ClearParameters();
		// ADD ANY PARAMETERS HERE
		_inst_fbParams.M_OutputToParameterList(_inst_arrParams);
		_inst_intStep := _inst_intStep + 10;
		
	20: // Route the command
		_bComplete := M_RouterHelper(
			_in_strMethodName := _strCOMMAND_NAME, 
			_in_timeTimeout := _timeCOMMAND_TIMEOUT,
			_inout_arrParams := _inst_arrParams,
			_inout_arrOutputs := _inst_arrOutputs,
			_out_strReturnValue=>_inst_strRet);
		
		// If route completed, move to next step
		IF _bComplete THEN
			_inst_intStep := _inst_intStep + 10;
			bRouterBusy := FALSE;
		ELSIF THIS^.P_bError THEN
			_inst_intStep := 0;
			bRouterBusy := FALSE;
		END_IF
		
	30: // Parse results
		_intRet := STRING_TO_INT(_inst_strRet);
		IF _intRet > 0 THEN
			_bResult := TRUE;
			THIS^.M_LogMessage(_strEND_MSG);
			// DO ANY PARSING HERE
			bConnected := TRUE;
		// Set error if command failed
		ELSE
			THIS^.M_SetError(_udintERROR_ID, _strERROR_MSG);
		END_IF
		// Go back to start
		_inst_intStep := 0;
END_CASE
M_StopMarking := _bResult;
intMStopMarkingStep := _inst_intStep;
END_METHOD

METHOD M_UpdateAllMarkingInformation : BOOL
VAR_INPUT
	MaxNumberOfBlocks	: INT;
//	MarkingInfo_Array	: ARRAY [0..255] OF OneBlockInfo;
END_VAR

VAR CONSTANT
	_strCOMMAND_NAME : T_MaxString	:= 'UpdateAllMarkingInformation'; // Name of the API method
	_timeCOMMAND_TIMEOUT : TIME		:= T#30S; // Max time to receive API response
	_strSTART_MSG : T_MaxString		:= 'UpdatingAllMarkingInformationInTheLaserProgram'; // Prints when method starts
	_strEND_MSG : T_MaxString		:= 'UpdatedAllMarkingInformationInTheLaserProgram'; // Prints when method finishes
	_udintERROR_ID : UDINT			:= KeyenceLaserMarkerMDX2000_Error.FailedToUpdateAllMarkingInformation; // Error ID to set if command fails
	_strERROR_MSG : T_MaxString		:= 'Failed to update All Marking Information in the Laser Marker program!'; // Error message to set if command fails
END_VAR

VAR_INST
	_inst_arrParams: T_ApiParameterList; // Parameters array
	_inst_arrOutputs: T_ApiParameterList; // Outputs array
	_inst_strRet: T_ApiParamValue; // Return string from the router
	_inst_intStep: INT; // Current method step
	_inst_fbParams: FB_ApiParamBuilder; // Parameter builder FB
END_VAR

VAR
	_bComplete: BOOL; // True if the routing finishes
	_intRet: INT; // Return string converted to an integer
	_bResult : BOOL; // Output of the method
	intIndex: INT;
	intIndex2 : INT;
	bOneTimeOnly : BOOL := TRUE;
END_VAR
_bResult := FALSE;
bMUpdateAllMarkingInfoBusy := TRUE;
_inst_intStep := intMUpdateAllMarkingInfoStep;
CASE _inst_intStep OF
	0: // Wait for no error and router not busy
		IF NOT THIS^.P_bError AND NOT bRouterBusy THEN
			bRouterBusy := TRUE;
			_inst_intStep := _inst_intStep + 10;
		END_IF
		
	10: // Initialize parameters
		THIS^.M_LogMessage(_strSTART_MSG);
		_inst_fbParams.M_ClearParameters();
		// ADD ANY PARAMETERS HERE
		_inst_fbParams.M_AddParameter('MaxNumberOfBlocks', MaxNumberOfBlocks);
		_inst_fbParams.M_OutputToParameterList(_inst_arrParams);
		_inst_intStep := _inst_intStep + 10;
		
	20: // Route the command
		_bComplete := M_RouterHelper(
			_in_strMethodName := _strCOMMAND_NAME, 
			_in_timeTimeout := _timeCOMMAND_TIMEOUT,
			_inout_arrParams := _inst_arrParams,
			_inout_arrOutputs := _inst_arrOutputs,
			_out_strReturnValue=>_inst_strRet);
		
		// If route completed, move to next step
		IF _bComplete THEN
			_inst_intStep := _inst_intStep + 10;
			bRouterBusy := FALSE;
		ELSIF THIS^.P_bError THEN
			_inst_intStep := 0;
			bRouterBusy := FALSE;
		END_IF
		
	30: // Parse results
		_intRet := STRING_TO_INT(_inst_strRet);
		IF _intRet > 0 THEN
			_bResult := TRUE;
			THIS^.M_LogMessage(_strEND_MSG);
			// DO ANY PARSING HERE
			_inst_fbParams.M_LoadFromParameterList(_inst_arrOutputs);
			bConnected := TRUE;
		// Set error if command failed
		ELSE
			THIS^.M_SetError(_udintERROR_ID, _strERROR_MSG);
		END_IF
		// Go back to start
		_inst_intStep := 0;
END_CASE
M_UpdateAllMarkingInformation := _bResult;
intMUpdateAllMarkingInfoStep := _inst_intStep;
END_METHOD

METHOD PUBLIC M_UpdateSingleBlockMarkingInformation : BOOL
VAR_INPUT
	BlockNumber : INT;
	BlockData : STRING;
	MarkEnabled : BOOL;
END_VAR

VAR CONSTANT
	_strCOMMAND_NAME : T_MaxString	:= 'UpdateSingleBlockMarkingInformation'; // Name of the API method
	_timeCOMMAND_TIMEOUT : TIME		:= T#30S; // Max time to receive API response
	_strSTART_MSG : T_MaxString		:= 'UpdatingSingleBlockMarkingInformationInTheLaserProgram'; // Prints when method starts
	_strEND_MSG : T_MaxString		:= 'UpdatedSingleBlockMarkingInformationInTheLaserProgram'; // Prints when method finishes
	_udintERROR_ID : UDINT			:= KeyenceLaserMarkerMDX2000_Error.FailedToUpdateSingleBlockMarkingInformation; // Error ID to set if command fails
	_strERROR_MSG : T_MaxString		:= 'Failed to update single block Marking Information in the Laser Marker program!'; // Error message to set if command fails
END_VAR

VAR_INST
	_inst_arrParams: T_ApiParameterList; // Parameters array
	_inst_arrOutputs: T_ApiParameterList; // Outputs array
	_inst_strRet: T_ApiParamValue; // Return string from the router
	_inst_intStep: INT; // Current method step
	_inst_fbParams: FB_ApiParamBuilder; // Parameter builder FB
END_VAR

VAR
	_bComplete: BOOL; // True if the routing finishes
	_intRet: INT; // Return string converted to an integer
	_bResult : BOOL; // Output of the method
	BlockType_INT : INT;
END_VAR
_bResult := FALSE;
bMUpdateSingleBlockInfoBusy := TRUE;
_inst_intStep := intMUpdateSingleBlockInfoStep;
CASE _inst_intStep OF
	0: // Wait for no error and router not busy
		IF NOT THIS^.P_bError AND NOT bRouterBusy THEN
			bRouterBusy := TRUE;
			_inst_intStep := _inst_intStep + 10;
		END_IF
		
	10: // Initialize parameters
		THIS^.M_LogMessage(_strSTART_MSG);
		_inst_fbParams.M_ClearParameters();
		// ADD ANY PARAMETERS HERE
		_inst_fbParams.M_AddParameter('BlockNumber', BlockNumber);
		_inst_fbParams.M_AddParameter('BlockData', BlockData);
		_inst_fbParams.M_AddParameter('MarkEnabled', MarkEnabled);
		_inst_fbParams.M_OutputToParameterList(_inst_arrParams);
		_inst_intStep := _inst_intStep + 10;
		
	20: // Route the command
		_bComplete := M_RouterHelper(
			_in_strMethodName := _strCOMMAND_NAME, 
			_in_timeTimeout := _timeCOMMAND_TIMEOUT,
			_inout_arrParams := _inst_arrParams,
			_inout_arrOutputs := _inst_arrOutputs,
			_out_strReturnValue=>_inst_strRet);
		
		// If route completed, move to next step
		IF _bComplete THEN
			_inst_intStep := _inst_intStep + 10;
			bRouterBusy := FALSE;
		ELSIF THIS^.P_bError THEN
			_inst_intStep := 0;
			bRouterBusy := FALSE;
		END_IF
		
	30: // Parse results
		_intRet := STRING_TO_INT(_inst_strRet);
		IF _intRet > 0 THEN
			_bResult := TRUE;
			THIS^.M_LogMessage(_strEND_MSG);
			// DO ANY PARSING HERE
			_inst_fbParams.M_LoadFromParameterList(_inst_arrOutputs);
			bConnected := TRUE;
		// Set error if command failed
		ELSE
			THIS^.M_SetError(_udintERROR_ID, _strERROR_MSG);
		END_IF
		// Go back to start
		_inst_intStep := 0;
END_CASE
M_UpdateSingleBlockMarkingInformation := _bResult;
intMUpdateSingleBlockInfoStep := _inst_intStep;
END_METHOD

(* This method should explicitly get the current program loaded on the device.
	If the current program is successfully gotten, this method should return
	TRUE and set P_strCurrentProgram and strCurrentProgram to the gotten
	program name. If this method fails, both should be set to empty strings. *)
METHOD M_GetCurrentProgram : BOOL
VAR_OUTPUT
	(* This should be set to the name of the currently loaded program if
		the method was successful, or a blank string otherwise. *)
	strCurrentProgram	: Sensata_Common.T_MaxString;
END_VAR
VAR CONSTANT
	_strCOMMAND_NAME : T_MaxString	:= 'GetCurrentProgram'; // Name of the API method
	_timeCOMMAND_TIMEOUT : TIME		:= T#45S; // Max time to receive API response
	_strSTART_MSG : T_MaxString		:= 'GettingCurrentProgramFromLaserMemory'; // Prints when method starts
	_strEND_MSG : T_MaxString		:= 'GotCurrentProgramFromLaserMemory'; // Prints when method finishes
	_udintERROR_ID : UDINT			:= KeyenceLaserMarkerMDX2000_Error.FailedToGetCurrentProgram; // Error ID to set if command fails
	_strERROR_MSG : T_MaxString		:= 'Failed to Get Current Laser Program from Laser Marker!'; // Error message to set if command fails
END_VAR

VAR_INST
	_inst_arrParams: T_ApiParameterList; // Parameters array
	_inst_arrOutputs: T_ApiParameterList; // Outputs array
	_inst_strRet: T_ApiParamValue; // Return string from the router
	_inst_intStep: INT; // Current method step
	_inst_fbParams: FB_ApiParamBuilder; // Parameter builder FB
END_VAR

VAR
	_bComplete: BOOL; // True if the routing finishes
	_intRet: INT; // Return string converted to an integer
	_bResult : BOOL; // Output of the method
END_VAR
_bResult := FALSE;
bMGetCurrentProgBusy := TRUE;
_inst_intStep := intMGetCurrentProgStep;
CASE _inst_intStep OF
	0: // Wait for no error and router not busy
		IF NOT THIS^.P_bError AND NOT bRouterBusy THEN
			bRouterBusy := TRUE;
			_inst_intStep := _inst_intStep + 10;
		END_IF
		
	10: // Initialize parameters
		THIS^.M_LogMessage(_strSTART_MSG);
		_inst_fbParams.M_ClearParameters();
		// ADD ANY PARAMETERS HERE
		_inst_fbParams.M_OutputToParameterList(_inst_arrParams);
		_inst_intStep := _inst_intStep + 10;
		
	20: // Route the command
		_bComplete := M_RouterHelper(
			_in_strMethodName := _strCOMMAND_NAME, 
			_in_timeTimeout := _timeCOMMAND_TIMEOUT,
			_inout_arrParams := _inst_arrParams,
			_inout_arrOutputs := _inst_arrOutputs,
			_out_strReturnValue=>_inst_strRet);
		
		// If route completed, move to next step
		IF _bComplete THEN
			_inst_intStep := _inst_intStep + 10;
			bRouterBusy := FALSE;
		ELSIF THIS^.P_bError THEN
			_inst_intStep := 0;
			bRouterBusy := FALSE;
		END_IF
		
	30: // Parse results
		_intRet := STRING_TO_INT(_inst_strRet);
		IF _intRet > 0 THEN
			_bResult := TRUE;
			THIS^.M_LogMessage(_strEND_MSG);
			// DO ANY PARSING HERE
			_inst_fbParams.M_LoadFromParameterList(_inst_arrOutputs);
			strCurrentProgram := _inst_fbParams.M_ParseString(_inst_fbParams.M_GetParameter('programName'));
			bConnected := TRUE;
		// Set error if command failed
		ELSE
			THIS^.M_SetError(_udintERROR_ID, _strERROR_MSG);
		END_IF
		// Go back to start
		_inst_intStep := 0;
END_CASE
M_GetCurrentProgram := _bResult;
intMGetCurrentProgStep := _inst_intStep;
END_METHOD

(* This method should explicitly check the program state of the device.
	Once the program state is known, this method should return TRUE and set
	P_enumProgramState and enumProgramState to the relevant E_ProgramState
	value, else it should set both to E_ProgramState.Unknown. *)
METHOD M_GetProgramState : BOOL
VAR_OUTPUT
	(* If the program state is successfully gotten, this should be set to
		the relevant E_ProgramState value. If this method fails, this should
		be set to E_ProgramState.Unknown. *)
	enumProgramState	: Sensata_Common.E_ProgramState;
END_VAR
M_GetProgramState := TRUE;
THIS^.M_LogWarning('M_GetProgramState is not implemented!');
END_METHOD

(* This method should load a new program onto the device, and then return TRUE
	once program loading is completed. Once this method begins the program loading
	process, P_strCurrentProgram should be cleared unless it is still explicitly
	known to be loaded. *)
METHOD M_LoadProgram : BOOL
VAR_INPUT
	(* String representing the program to load. If string must be in a specific
		format, make sure to override this comment to document it. *)
	//strProgram	: Sensata_Common.T_MaxString;
	
	//Replace filepath with just program number and also 
//	filepath : STRING;	// filepath where the program is stored
//	LaserMemoryLocation : INT; // Laser Memory location where the program needs to be loaded 
	
END_VAR

VAR CONSTANT
	_strCOMMAND_NAME : T_MaxString	:= 'LoadProgram'; // Name of the API method
	_timeCOMMAND_TIMEOUT : TIME		:= T#30S; // Max time to receive API response
	_strSTART_MSG : T_MaxString		:= 'LoadingProgramToLaser'; // Prints when method starts
	_strEND_MSG : T_MaxString		:= 'ProgramLoadedToLaser'; // Prints when method finishes
	_udintERROR_ID : UDINT			:= KeyenceLaserMarkerMDX2000_Error.FailedToSendProgramToLaser; // Error ID to set if command fails
	_strERROR_MSG : T_MaxString		:= 'Failed to Load Program to Laser Marker!'; // Error message to set if command fails
END_VAR

VAR_INST
	_inst_arrParams: T_ApiParameterList; // Parameters array
	_inst_arrOutputs: T_ApiParameterList; // Outputs array
	_inst_strRet: T_ApiParamValue; // Return string from the router
	_inst_intStep: INT; // Current method step
	_inst_fbParams: FB_ApiParamBuilder; // Parameter builder FB
END_VAR

VAR
	_bComplete: BOOL; // True if the routing finishes
	_intRet: INT; // Return string converted to an integer
	_bResult : BOOL; // Output of the method	
END_VAR
_bResult := FALSE;
bMLoadProgramBusy := TRUE;
_inst_intStep := intMLoadProgramStep;
CASE _inst_intStep OF
	0: // Wait for no error and router not busy
		IF NOT THIS^.P_bError AND NOT bRouterBusy THEN
			bRouterBusy := TRUE;
			_inst_intStep := _inst_intStep + 10;
		END_IF
		
	10: // Initialize parameters
		THIS^.M_LogMessage(_strSTART_MSG);
		_inst_fbParams.M_ClearParameters();
		// ADD ANY PARAMETERS HERE
		_inst_fbParams.M_AddParameter('programName', in_strProgram);
		_inst_fbParams.M_OutputToParameterList(_inst_arrParams);
		_inst_intStep := _inst_intStep + 10;
		
	20: // Route the command
		_bComplete := M_RouterHelper(
			_in_strMethodName := _strCOMMAND_NAME, 
			_in_timeTimeout := _timeCOMMAND_TIMEOUT,
			_inout_arrParams := _inst_arrParams,
			_inout_arrOutputs := _inst_arrOutputs,
			_out_strReturnValue=>_inst_strRet);
		
		// If route completed, move to next step
		IF _bComplete THEN
			_inst_intStep := _inst_intStep + 10;
			bRouterBusy := FALSE;
		ELSIF THIS^.P_bError THEN
			_inst_intStep := 0;
			bRouterBusy := FALSE;
		END_IF
		
	30: // Parse results
		_intRet := STRING_TO_INT(_inst_strRet);
		IF _intRet > 0 THEN
			_bResult := TRUE;
			THIS^.M_LogMessage(_strEND_MSG);
			// DO ANY PARSING HERE
		// Set error if command failed
		ELSE
			THIS^.M_SetError(_udintERROR_ID, _strERROR_MSG);
		END_IF
		// Go back to start
		_inst_intStep := 0;
END_CASE
M_LoadProgram := _bResult;
intMLoadProgramStep := _inst_intStep;
END_METHOD

(* This program should move to the program state from whatever state it was in
	to the Paused state, and then return TRUE once successful. If the program
	state is Stopped, this method should return TRUE but keep the current state
	as Stopped, since Paused at the beginning at the program is equivalent to
	being Stopped. *)
METHOD M_PauseProgram : BOOL
M_PauseProgram := TRUE;
THIS^.M_LogWarning('M_PauseProgram is not implemented!');
END_METHOD

METHOD PUBLIC M_SaveCurrentLaserProgramtoPC : BOOL
VAR_INPUT
	LaserProgramFolderPath : STRING;
END_VAR
VAR_OUTPUT
	out_bool_SaveProgramToPC_Success : BOOL;
END_VAR
VAR CONSTANT
	_strCOMMAND_NAME : T_MaxString	:= 'SaveCurrentLaserProgramToPC'; // Name of the API method
	_timeCOMMAND_TIMEOUT : TIME		:= T#45S; // Max time to receive API response
	_strSTART_MSG : T_MaxString		:= 'SavingCurrentProgram'; // Prints when method starts
	_strEND_MSG : T_MaxString		:= 'SavedCurrentProgram'; // Prints when method finishes
	_udintERROR_ID : UDINT			:= KeyenceLaserMarkerMDX2000_Error.FailedToSaveCurrentLaserProgramToPC; // Error ID to set if command fails
	_strERROR_MSG : T_MaxString		:= 'Failed to Save Current Laser Program to PC from Laser Marker!'; // Error message to set if command fails
END_VAR

VAR_INST
	_inst_arrParams: T_ApiParameterList; // Parameters array
	_inst_arrOutputs: T_ApiParameterList; // Outputs array
	_inst_strRet: T_ApiParamValue; // Return string from the router
	_inst_intStep: INT; // Current method step
	_inst_fbParams: FB_ApiParamBuilder; // Parameter builder FB
END_VAR

VAR
	_bComplete: BOOL; // True if the routing finishes
	_intRet: INT; // Return string converted to an integer
	_bResult : BOOL; // Output of the method
END_VAR
_bResult := FALSE;
bMSaveCurrentLaserProgramtoPCBusy := TRUE;
_inst_intStep := intMSaveCurrentLaserProgramtoPC;
CASE _inst_intStep OF
	0: // Wait for no error and router not busy
		IF NOT THIS^.P_bError AND NOT bRouterBusy THEN
			bRouterBusy := TRUE;
			_inst_intStep := _inst_intStep + 10;
		END_IF
		
	10: // Initialize parameters
		THIS^.M_LogMessage(_strSTART_MSG);
		_inst_fbParams.M_ClearParameters();
		// ADD ANY PARAMETERS HERE
		_inst_fbParams.M_AddParameter('LaserProgramFolderPath',LaserProgramFolderPath);
		_inst_fbParams.M_OutputToParameterList(_inst_arrParams);
		_inst_intStep := _inst_intStep + 10;
		
	20: // Route the command
		_bComplete := M_RouterHelper(
			_in_strMethodName := _strCOMMAND_NAME, 
			_in_timeTimeout := _timeCOMMAND_TIMEOUT,
			_inout_arrParams := _inst_arrParams,
			_inout_arrOutputs := _inst_arrOutputs,
			_out_strReturnValue=>_inst_strRet);
		
		// If route completed, move to next step
		IF _bComplete THEN
			_inst_intStep := _inst_intStep + 10;
			bRouterBusy := FALSE;
		ELSIF THIS^.P_bError THEN
			_inst_intStep := 0;
			bRouterBusy := FALSE;
		END_IF
		
	30: // Parse results
		_intRet := STRING_TO_INT(_inst_strRet);
		IF _intRet > 0 THEN
			_bResult := TRUE;
			THIS^.M_LogMessage(_strEND_MSG);
			// DO ANY PARSING HERE
			_inst_fbParams.M_LoadFromParameterList(_inst_arrOutputs);
			out_bool_SaveProgramToPC_Success := _inst_fbParams.M_ParseBool(_inst_fbParams.M_GetParameter('out_bool_SaveProgramToPC_Success'));
			bConnected := TRUE;
		// Set error if command failed
		ELSE
			THIS^.M_SetError(_udintERROR_ID, _strERROR_MSG);
		END_IF
		// Go back to start
		_inst_intStep := 0;
END_CASE
M_SaveCurrentLaserProgramtoPC := _bResult;
intMSaveCurrentLaserProgramtoPC := _inst_intStep;
END_METHOD

METHOD PUBLIC M_SendProgramtoLaser : BOOL
VAR_INPUT
	filepath : STRING;	// filepath where the program is stored
	LaserMemoryLocation : INT; // Laser Memory location where the program needs to be loaded 
END_VAR

VAR_OUTPUT
	out_bool_SendProgramToLaserSuccess : BOOL;
END_VAR

VAR CONSTANT
	_strCOMMAND_NAME : T_MaxString	:= 'SendProgramtoLaser'; // Name of the API method
	_timeCOMMAND_TIMEOUT : TIME		:= T#30S; // Max time to receive API response
	_strSTART_MSG : T_MaxString		:= 'SendingProgramToLaser'; // Prints when method starts
	_strEND_MSG : T_MaxString		:= 'SentProgramToLaser'; // Prints when method finishes
	_udintERROR_ID : UDINT			:= KeyenceLaserMarkerMDX2000_Error.FailedToSendProgramToLaser; // Error ID to set if command fails
	_strERROR_MSG : T_MaxString		:= 'Failed to Send Program to Laser Marker!'; // Error message to set if command fails
END_VAR

VAR_INST
	_inst_arrParams: T_ApiParameterList; // Parameters array
	_inst_arrOutputs: T_ApiParameterList; // Outputs array
	_inst_strRet: T_ApiParamValue; // Return string from the router
	_inst_intStep: INT; // Current method step
	_inst_fbParams: FB_ApiParamBuilder; // Parameter builder FB
END_VAR

VAR
	_bComplete: BOOL; // True if the routing finishes
	_intRet: INT; // Return string converted to an integer
	_bResult : BOOL; // Output of the method	

END_VAR
_bResult := FALSE;
bMSendProgramToLaserBusy := TRUE;
_inst_intStep := intMSendProgramToLaserStep;
CASE _inst_intStep OF
	0: // Wait for no error and router not busy
		IF NOT THIS^.P_bError AND NOT bRouterBusy THEN
			bRouterBusy := TRUE;
			_inst_intStep := _inst_intStep + 10;
		END_IF
		
	10: // Initialize parameters
		THIS^.M_LogMessage(_strSTART_MSG);
		_inst_fbParams.M_ClearParameters();
		// ADD ANY PARAMETERS HERE
		_inst_fbParams.M_AddParameter('filepath', filepath);
		_inst_fbParams.M_AddParameter('LaserMemoryLocation', LaserMemoryLocation);
		_inst_fbParams.M_OutputToParameterList(_inst_arrParams);
		_inst_intStep := _inst_intStep + 10;
		
	20: // Route the command
		_bComplete := M_RouterHelper(
			_in_strMethodName := _strCOMMAND_NAME, 
			_in_timeTimeout := _timeCOMMAND_TIMEOUT,
			_inout_arrParams := _inst_arrParams,
			_inout_arrOutputs := _inst_arrOutputs,
			_out_strReturnValue=>_inst_strRet);
		
		// If route completed, move to next step
		IF _bComplete THEN
			_inst_intStep := _inst_intStep + 10;
			bRouterBusy := FALSE;
		ELSIF THIS^.P_bError THEN
			_inst_intStep := 0;
			bRouterBusy := FALSE;
		END_IF
		
	30: // Parse results
		_intRet := STRING_TO_INT(_inst_strRet);
		IF _intRet > 0 THEN
			_bResult := TRUE;
			THIS^.M_LogMessage(_strEND_MSG);
			// DO ANY PARSING HERE
			_inst_fbParams.M_LoadFromParameterList(_inst_arrOutputs);
			out_bool_SendProgramToLaserSuccess := _inst_fbParams.M_ParseBool(_inst_fbParams.M_GetParameter('out_bool_SendProgramToLaserSuccess'));
			bConnected := TRUE;
		// Set error if command failed
		ELSE
			THIS^.M_SetError(_udintERROR_ID, _strERROR_MSG);
		END_IF
		// Go back to start
		_inst_intStep := 0;
END_CASE
M_SendProgramtoLaser := _bResult;
intMSendProgramToLaserStep := _inst_intStep;
END_METHOD

(* This should move the program state from whatever state it is in to the
	Running state, and then return TRUE once successful. Starting from the
	Paused state should always continue execution from whatever point the
	program was at when the program was initially paused. *)
METHOD M_StartProgram : BOOL
M_StartProgram := TRUE;
THIS^.M_LogWarning('M_StartProgram is not implemented!');
END_METHOD

(* This should change the program state from whatever state it was in to the
	Stopped state and then return TRUE. Moving to the Stopped state should
	always reset the program execution back to the beginning. *)
METHOD M_StopProgram : BOOL
M_StopProgram := TRUE;
THIS^.M_LogWarning('M_StopProgram is not implemented!');
END_METHOD

METHOD PUBLIC M_UpdateSingleProgramBlockData : BOOL
VAR_INPUT
	LaserProgramMemoryLocation : INT;
	BlockNumber : INT;
	BlockData : STRING;
	BlockType : BlockTypes;
END_VAR
VAR_OUTPUT
	out_bool_UpdateData_Success : BOOL;
END_VAR
VAR CONSTANT
	_strCOMMAND_NAME : T_MaxString	:= 'UpdateSingleBlockData'; // Name of the API method
	_timeCOMMAND_TIMEOUT : TIME		:= T#30S; // Max time to receive API response
	_strSTART_MSG : T_MaxString		:= 'UpdatingSingleBlockdataInTheLaserProgram'; // Prints when method starts
	_strEND_MSG : T_MaxString		:= 'UpdatedSingleBlockdataInTheLaserProgram'; // Prints when method finishes
	_udintERROR_ID : UDINT			:= KeyenceLaserMarkerMDX2000_Error.FailedToUpdateSingleBlockData; // Error ID to set if command fails
	_strERROR_MSG : T_MaxString		:= 'Failed to update single block data in the Laser Marker program!'; // Error message to set if command fails
END_VAR

VAR_INST
	_inst_arrParams: T_ApiParameterList; // Parameters array
	_inst_arrOutputs: T_ApiParameterList; // Outputs array
	_inst_strRet: T_ApiParamValue; // Return string from the router
	_inst_intStep: INT; // Current method step
	_inst_fbParams: FB_ApiParamBuilder; // Parameter builder FB
END_VAR

VAR
	_bComplete: BOOL; // True if the routing finishes
	_intRet: INT; // Return string converted to an integer
	_bResult : BOOL; // Output of the method
	BlockType_INT : INT;
END_VAR
_bResult := FALSE;
bMUpdateSingleProgramBlockDataBusy := TRUE;
_inst_intStep := intMUpdateSingleProgramBlockDataStep;
CASE _inst_intStep OF
	0: // Wait for no error and router not busy
		IF NOT THIS^.P_bError AND NOT bRouterBusy THEN
			bRouterBusy := TRUE;
			_inst_intStep := _inst_intStep + 10;
		END_IF
		
	10: // Initialize parameters
		THIS^.M_LogMessage(_strSTART_MSG);
		_inst_fbParams.M_ClearParameters();
		// ADD ANY PARAMETERS HERE
		BlockType_INT := TO_INT(BlockType);
		_inst_fbParams.M_AddParameter('LaserProgramMemoryLocation', LaserProgramMemoryLocation);
		_inst_fbParams.M_AddParameter('BlockNumber', BlockNumber);
		_inst_fbParams.M_AddParameter('BlockData', BlockData);
		_inst_fbParams.M_AddParameter('BlockType', BlockType_INT);
		_inst_fbParams.M_OutputToParameterList(_inst_arrParams);
		_inst_intStep := _inst_intStep + 10;
		
	20: // Route the command
		_bComplete := M_RouterHelper(
			_in_strMethodName := _strCOMMAND_NAME, 
			_in_timeTimeout := _timeCOMMAND_TIMEOUT,
			_inout_arrParams := _inst_arrParams,
			_inout_arrOutputs := _inst_arrOutputs,
			_out_strReturnValue=>_inst_strRet);
		
		// If route completed, move to next step
		IF _bComplete THEN
			_inst_intStep := _inst_intStep + 10;
			bRouterBusy := FALSE;
		ELSIF THIS^.P_bError THEN
			_inst_intStep := 0;
			bRouterBusy := FALSE;
		END_IF
		
	30: // Parse results
		_intRet := STRING_TO_INT(_inst_strRet);
		IF _intRet > 0 THEN
			_bResult := TRUE;
			THIS^.M_LogMessage(_strEND_MSG);
			// DO ANY PARSING HERE
			_inst_fbParams.M_LoadFromParameterList(_inst_arrOutputs);
			out_bool_UpdateData_Success := _inst_fbParams.M_ParseBool(_inst_fbParams.M_GetParameter('out_bool_UpdateData_Success'));
			bConnected := TRUE;
		// Set error if command failed
		ELSE
			THIS^.M_SetError(_udintERROR_ID, _strERROR_MSG);
		END_IF
		// Go back to start
		_inst_intStep := 0;
END_CASE
M_UpdateSingleProgramBlockData := _bResult;
intMUpdateSingleProgramBlockDataStep := _inst_intStep;
END_METHOD

METHOD PUBLIC M_UpdateSingleProgramBlockMarkEnabled : BOOL
VAR_INPUT
	LaserProgramMemoryLocation : INT;
	BlockNumber : INT;
	BlockType : BlockTypes;
	MarkEnabled : BOOL;
	//int LaserProgramMemoryLocation, int BlockNumber, bool MarkEnabled, BlockTypes BlockType, out bool out_bool_UpdateSingleBlockMarkEnabledIntheLaser_Success
END_VAR
VAR_OUTPUT
	out_bool_MarkEnabled_Success : BOOL;
END_VAR
VAR CONSTANT
	_strCOMMAND_NAME : T_MaxString	:= 'UpdateSingleBlockMarkEnabled'; // Name of the API method
	_timeCOMMAND_TIMEOUT : TIME		:= T#30S; // Max time to receive API response
	_strSTART_MSG : T_MaxString		:= 'UpdatingSingleBlockMarkEnabledStatusInTheLaserProgram'; // Prints when method starts
	_strEND_MSG : T_MaxString		:= 'UpdatedSingleBlockMarkEnabledStatusInTheLaserProgram'; // Prints when method finishes
	_udintERROR_ID : UDINT			:= KeyenceLaserMarkerMDX2000_Error.FailedToUpdateSingleBlockMarkEnabledProperty; // Error ID to set if command fails
	_strERROR_MSG : T_MaxString		:= 'Failed to update single block mark enabled status in the Laser Marker program!'; // Error message to set if command fails
END_VAR

VAR_INST
	_inst_arrParams: T_ApiParameterList; // Parameters array
	_inst_arrOutputs: T_ApiParameterList; // Outputs array
	_inst_strRet: T_ApiParamValue; // Return string from the router
	_inst_intStep: INT; // Current method step
	_inst_fbParams: FB_ApiParamBuilder; // Parameter builder FB
END_VAR

VAR
	_bComplete: BOOL; // True if the routing finishes
	_intRet: INT; // Return string converted to an integer
	_bResult : BOOL; // Output of the method
	_dummy_pointer : PVOID;
	BlockType_INT : INT;
END_VAR
_bResult := FALSE;
bMUpdateSingleProgramBlockMarkingEnabledBusy := TRUE;
_inst_intStep := intMUpdateSingleProgramBlockMarkingEnabledStep;
CASE _inst_intStep OF
	0: // Wait for no error and router not busy
		IF NOT THIS^.P_bError AND NOT bRouterBusy THEN
			bRouterBusy := TRUE;
			_inst_intStep := _inst_intStep + 10;
		END_IF
		
	10: // Initialize parameters
		THIS^.M_LogMessage(_strSTART_MSG);
		_inst_fbParams.M_ClearParameters();
		// ADD ANY PARAMETERS HERE
		BlockType_INT := TO_INT(BlockType);
		_inst_fbParams.M_AddParameter('LaserProgramMemoryLocation', LaserProgramMemoryLocation);
		_inst_fbParams.M_AddParameter('BlockNumber', BlockNumber);
		_inst_fbParams.M_AddParameter('MarkEnabled', MarkEnabled);
		_inst_fbParams.M_AddParameter('BlockType', BlockType_INT);
		_inst_fbParams.M_OutputToParameterList(_inst_arrParams);
		_inst_intStep := _inst_intStep + 10;
		
	20: // Route the command
		_bComplete := M_RouterHelper(
			_in_strMethodName := _strCOMMAND_NAME, 
			_in_timeTimeout := _timeCOMMAND_TIMEOUT,
			_inout_arrParams := _inst_arrParams,
			_inout_arrOutputs := _inst_arrOutputs,
			_out_strReturnValue=>_inst_strRet);
		
		// If route completed, move to next step
		IF _bComplete THEN
			_inst_intStep := _inst_intStep + 10;
			bRouterBusy := FALSE;
		ELSIF THIS^.P_bError THEN
			_inst_intStep := 0;
			bRouterBusy := FALSE;
		END_IF
		
	30: // Parse results
		_intRet := STRING_TO_INT(_inst_strRet);
		IF _intRet > 0 THEN
			_bResult := TRUE;
			THIS^.M_LogMessage(_strEND_MSG);
			// DO ANY PARSING HERE
			_inst_fbParams.M_LoadFromParameterList(_inst_arrOutputs);
			out_bool_MarkEnabled_Success := _inst_fbParams.M_ParseBool(_inst_fbParams.M_GetParameter('out_bool_MarkEnabled_Success'));
			bConnected := TRUE;
		// Set error if command failed
		ELSE
			THIS^.M_SetError(_udintERROR_ID, _strERROR_MSG);
		END_IF
		// Go back to start
		_inst_intStep := 0;
END_CASE
M_UpdateSingleProgramBlockMarkEnabled := _bResult;
intMUpdateSingleProgramBlockMarkingEnabledStep := _inst_intStep;
END_METHOD

(* This property should be TRUE while any method in this interface is actively
	executing, or FALSE otherwise. *)
PROPERTY P_bProgramControlBusy : BOOL
GET
END_GET
END_PROPERTY

(* The current E_ProgramState value of the device. This should be reset to
	E_ProgramState.Unknown if any methods in this interface interact with the
	device but fail. *)
PROPERTY P_enumProgramState : Sensata_Common.E_ProgramState
GET
END_GET
END_PROPERTY

(* The value of the currently loaded program. This should only be set by
	M_LoadProgram or M_GetCurrentProgram, and set to a blank string if either
	fail. *)
PROPERTY P_strCurrentProgram : Sensata_Common.T_MaxString
GET
END_GET
END_PROPERTY

METHOD PUBLIC M_GetLaserActivatedStatus : BOOL
VAR_INPUT
//	LaserProgramFolderPath : STRING;
END_VAR
VAR_OUTPUT
	out_IsLaserActivated : BOOL;
END_VAR
VAR CONSTANT
	_strCOMMAND_NAME : T_MaxString	:= 'GetLaserActivatedStatus'; // Name of the API method
	_timeCOMMAND_TIMEOUT : TIME		:= T#30S; // Max time to receive API response
	_strSTART_MSG : T_MaxString		:= 'GettingLaserActivatedStatus'; // Prints when method starts
	_strEND_MSG : T_MaxString		:= 'ReceivedLaserActivatedStatus'; // Prints when method finishes
	_udintERROR_ID : UDINT			:= KeyenceLaserMarkerMDX2000_Error.FailedToGetLaserActivatedStatus; // Error ID to set if command fails
	_strERROR_MSG : T_MaxString		:= 'Failed to Get Laser Activated Status from Laser Marker!'; // Error message to set if command fails
END_VAR

VAR_INST
	_inst_arrParams: T_ApiParameterList; // Parameters array
	_inst_arrOutputs: T_ApiParameterList; // Outputs array
	_inst_strRet: T_ApiParamValue; // Return string from the router
	_inst_intStep: INT; // Current method step
	_inst_fbParams: FB_ApiParamBuilder; // Parameter builder FB
END_VAR

